(*=======================================================*)
	170:	(* WT Nummer schreiben *)
		IF	 fb_state_entry.E THEN
			(* Starte Schreib Prozess *)
			balluff_tag_reader.fb.i16_addresse := 0;
			balluff_tag_reader.fb.i16_anzahl_byte := 1;
			balluff_tag_reader.fb.s_schreib_daten[0] := gst_tag_data.WpcNumber;
			balluff_tag_reader.st_ctrl.in.b_start_schreiben := TRUE;
		END_IF

		(*-----------------------Weiterschaltbedingungen----------------------------*)
		IF 	balluff_tag_reader.st_ctrl.out.b_fertig AND NOT fb_state_entry.E THEN
			balluff_tag_reader.st_ctrl.in.b_start_schreiben := FALSE;
			fb_state_entry.i16_next_step := 180;
		END_IF

(*=======================================================*)
	180:	(* letztes benutzes Werkzeug schreiben*)
		IF 	fb_state_entry.E THEN
			(* Starte Schreib Prozess *)
			IF gst_datensatz.st_md.i16_tag_data_structur_version = 0 THEN
				balluff_tag_reader.fb.i16_addresse := 54;
				balluff_tag_reader.fb.i16_anzahl_byte := 1;
				balluff_tag_reader.fb.s_schreib_daten[0] := gst_tag_data.LastUsedTool;
				balluff_tag_reader.st_ctrl.in.b_start_schreiben := TRUE;
			ELSIF gst_datensatz.st_md.i16_tag_data_structur_version = 1 THEN
				balluff_tag_reader.fb.i16_addresse := 15;
				balluff_tag_reader.fb.i16_anzahl_byte := 1;
				balluff_tag_reader.fb.s_schreib_daten[0] := gst_tag_data.LastUsedTool;
				balluff_tag_reader.st_ctrl.in.b_start_schreiben := TRUE;
			END_IF
		END_IF

		(*-----------------------Weiterschaltbedingungen----------------------------*)
		IF 	balluff_tag_reader.st_ctrl.out.b_fertig AND NOT fb_state_entry.E THEN
			balluff_tag_reader.st_ctrl.in.b_start_schreiben := FALSE;
			IF gst_datensatz.st_md.i16_tag_data_structur_version = 0 THEN
				fb_state_entry.i16_next_step := 120;
			ELSIF gst_datensatz.st_md.i16_tag_data_structur_version = 1 THEN
				fb_state_entry.i16_next_step := 190;
			END_IF
		END_IF

(*=======================================================*)
	190:	(* Anzahl ISK auf WT *)
		IF 	fb_state_entry.E THEN
			(* Starte Schreib Prozess *)
			balluff_tag_reader.fb.i16_addresse := 10;
			balluff_tag_reader.fb.i16_anzahl_byte := 1;
			balluff_tag_reader.fb.s_schreib_daten[0] := gst_tag_data.AmountPartsOnWpc;
			balluff_tag_reader.st_ctrl.in.b_start_schreiben := TRUE;
		END_IF

		(*-----------------------Weiterschaltbedingungen----------------------------*)
		IF 	balluff_tag_reader.st_ctrl.out.b_fertig AND NOT fb_state_entry.E THEN
			balluff_tag_reader.st_ctrl.in.b_start_schreiben := FALSE;
			fb_state_entry.i16_next_step := 120;
		END_IF

(*=======================================================*)
	200:	(*WT zurücksetzen*)
		IF	 fb_state_entry.E THEN
			IF gst_datensatz.st_md.i16_tag_data_structur_version = 0 THEN
				gst_tag_data.StateParts[0] := PART_NO;
				gst_tag_data.StateParts[1] := PART_NO;

				balluff_tag_reader.st_ctrl.in.b_start_schreiben := TRUE;
				balluff_tag_reader.fb.i16_addresse := 1;
				balluff_tag_reader.fb.i16_anzahl_byte := 2;
				balluff_tag_reader.fb.s_schreib_daten[0] := DINT_TO_BYTE(gst_tag_data.StateParts[0]);
				balluff_tag_reader.fb.s_schreib_daten[1] := DINT_TO_BYTE(gst_tag_data.StateParts[1]);
			ELSIF gst_datensatz.st_md.i16_tag_data_structur_version = 1 THEN
				FOR i:= 0 TO 7 BY 1 DO
					gst_tag_data.StateParts[i] := PART_NO;
				END_FOR
	
				balluff_tag_reader.st_ctrl.in.b_start_schreiben := TRUE;
				balluff_tag_reader.fb.i16_addresse := 1;
				balluff_tag_reader.fb.i16_anzahl_byte := 8;
				FOR i:= 0 TO 7 BY 1 DO
					balluff_tag_reader.fb.s_schreib_daten[i] := DINT_TO_BYTE(gst_tag_data.StateParts[i]);
				END_FOR
			END_IF
		END_IF

		(*-----------------------Weiterschaltbedingungen----------------------------*)
		IF 	balluff_tag_reader.st_ctrl.out.b_fertig AND NOT fb_state_entry.E THEN
			(* Ok: Daten sind auf dem Tag *)
			balluff_tag_reader.st_ctrl.in.b_start_schreiben := FALSE;
			fb_state_entry.i16_next_step := 210;
		END_IF

(*=======================================================*)
	210:	(* letztes benutzes Werkzeug schreiben*)
		IF 	fb_state_entry.E THEN
			gst_tag_data.LastUsedTool := 0;
			(* Starte Schreib Prozess *)
			IF gst_datensatz.st_md.i16_tag_data_structur_version = 0 THEN
				balluff_tag_reader.fb.i16_addresse := 54;
				balluff_tag_reader.fb.i16_anzahl_byte := 1;
				balluff_tag_reader.fb.s_schreib_daten[0] := 0;
				balluff_tag_reader.st_ctrl.in.b_start_schreiben := TRUE;
			ELSIF gst_datensatz.st_md.i16_tag_data_structur_version = 1 THEN
				balluff_tag_reader.fb.i16_addresse := 15;
				balluff_tag_reader.fb.i16_anzahl_byte := 1;
				balluff_tag_reader.fb.s_schreib_daten[0] := 0;
				balluff_tag_reader.st_ctrl.in.b_start_schreiben := TRUE;
			END_IF
		END_IF

		(*-----------------------Weiterschaltbedingungen----------------------------*)
		IF 	balluff_tag_reader.st_ctrl.out.b_fertig AND NOT fb_state_entry.E THEN
			balluff_tag_reader.st_ctrl.in.b_start_schreiben := FALSE;
			fb_state_entry.i16_next_step := INIT;
		END_IF

(*=======================================================*)
	FEHLER:
		IF 	fb_state_entry.E THEN
			st_ctrl_out.b_fehler := TRUE;
			fb_ton_quitt.IN := FALSE;
		END_IF

		(*-----------------------Weiterschaltbedingungen----------------------------*)
		IF 	st_ctrl_in.b_quitt AND NOT fb_state_entry.E THEN
			st_ctrl_out.b_fehler := FALSE;
			fb_ton_quitt.IN := TRUE;
		END_IF

		IF 	fb_ton_quitt.Q THEN
			fb_ton_quitt.IN := FALSE;
			fb_state_entry.i16_next_step := INIT;
		END_IF

(*=======================================================*)
	STOP:
		IF 	fb_state_entry.E THEN
			;
		END_IF

		(*-----------------------Weiterschaltbedingungen----------------------------*)
		IF 	Balluff_Tag_Reader.fb.fb_state_entry.i16_step=BEREIT THEN
			fb_state_entry.i16_next_step := INIT;
		END_IF

END_CASE

fb_state_entry(
	i16_next_step:= ,
	i16_pos:= 2,
	s_debugtext:= ,
	E=> ,
	X=> ,
	i16_step=> ,
	i16_last_step=> );

(* Fehlermeldungen ab dem Startindex in das globale Störmeldungsarray schreiben *)
garr_stoermeldungen[st_config.i16_meld_startindex + 0] := sm_WT_Nummer_ungueltig;
garr_stoermeldungen[st_config.i16_meld_startindex + 1] := sm_wt_hat_kein_tag;
garr_stoermeldungen[st_config.i16_meld_startindex + 2] :=FALSE;
garr_stoermeldungen[st_config.i16_meld_startindex + 3] := FALSE;
garr_stoermeldungen[st_config.i16_meld_startindex + 4] := FALSE;
garr_stoermeldungen[st_config.i16_meld_startindex + 5] := FALSE;
garr_stoermeldungen[st_config.i16_meld_startindex + 6] := FALSE;
garr_stoermeldungen[st_config.i16_meld_startindex + 7] := FALSE;
garr_stoermeldungen[st_config.i16_meld_startindex + 8] := FALSE;
garr_stoermeldungen[st_config.i16_meld_startindex + 9] := FALSE;
garr_stoermeldungen[st_config.i16_meld_startindex + 10] := FALSE;
garr_stoermeldungen[st_config.i16_meld_startindex + 11] := FALSE;
garr_stoermeldungen[st_config.i16_meld_startindex + 12] := FALSE;
garr_stoermeldungen[st_config.i16_meld_startindex + 13] := FALSE;
garr_stoermeldungen[st_config.i16_meld_startindex + 14] := FALSE;
garr_stoermeldungen[st_config.i16_meld_startindex + 15] := FALSE;
garr_stoermeldungen[st_config.i16_meld_startindex + 16] := FALSE;
garr_stoermeldungen[st_config.i16_meld_startindex + 17] := FALSE;
garr_stoermeldungen[st_config.i16_meld_startindex + 18] := FALSE;
garr_stoermeldungen[st_config.i16_meld_startindex + 19] := FALSE;

garr_betriebsmeldungen[st_config.i16_meld_startindex + 0] := bm_kein_WT_im_Aktionsfeld;
garr_betriebsmeldungen[st_config.i16_meld_startindex + 1] := bm_Wert_nicht_erlaubt;
garr_betriebsmeldungen[st_config.i16_meld_startindex + 2] := FALSE;
garr_betriebsmeldungen[st_config.i16_meld_startindex + 3] := FALSE;
garr_betriebsmeldungen[st_config.i16_meld_startindex + 4] := FALSE;
garr_betriebsmeldungen[st_config.i16_meld_startindex + 5] := FALSE;
garr_betriebsmeldungen[st_config.i16_meld_startindex + 6] := FALSE;
garr_betriebsmeldungen[st_config.i16_meld_startindex + 7] := FALSE;
garr_betriebsmeldungen[st_config.i16_meld_startindex + 8] := FALSE;
garr_betriebsmeldungen[st_config.i16_meld_startindex + 9] := FALSE;
garr_betriebsmeldungen[st_config.i16_meld_startindex + 10] := FALSE;
garr_betriebsmeldungen[st_config.i16_meld_startindex + 11] := FALSE;
garr_betriebsmeldungen[st_config.i16_meld_startindex + 12] := FALSE;
garr_betriebsmeldungen[st_config.i16_meld_startindex + 13] := FALSE;
garr_betriebsmeldungen[st_config.i16_meld_startindex + 14] := FALSE;
garr_betriebsmeldungen[st_config.i16_meld_startindex + 15] := FALSE;
garr_betriebsmeldungen[st_config.i16_meld_startindex + 16] := FALSE;
garr_betriebsmeldungen[st_config.i16_meld_startindex + 17] := FALSE;
garr_betriebsmeldungen[st_config.i16_meld_startindex + 18] := FALSE;
garr_betriebsmeldungen[st_config.i16_meld_startindex + 19] := FALSE;
END_PROGRAM

(* POU Gemeinsamkeiten17xx/Bandeinzug/ST_Anwahl_Bandeinzug, ST *)
PROGRAM ST_Anwahl_Bandeinzug
VAR
	b_first_cycle 						: BOOL := TRUE;
	i16_typ_bandeinzug_visu			: enum_typ_bandeinzug_visu := KEIN_BANDEINZUG;
END_VAR
(*======================================================
   PRG: ExportResultString
 ------------------------------------------------------
   Auth: 		Werner Friedl    						 
   Date: 		07.03.2016    						     
   Rev.: 		1.0	
   Desc:		Damit bei unterschiedlichen Zellen (1700 oder 1720) nur die vorhandenen Bandwechsler in der Visu vorne angezeigt werden,
			müssen diese der Struktur "i16_typ_bandeinzug" zugewiesen werden.
   Historie:   1.0

 ========================================================*)
IF 	gi16_bbgen_auftrag = LESE_WKZ THEN
	b_first_cycle:=TRUE;
END_IF



IF	NOT b_first_cycle THEN

	CASE gst_datensatz.st_md.i16_typ_zelle OF
		KEINE_ZELLE:
			;

		BESTUECKZELLE_1700, RASTERFOLIE:
	
			CASE i16_typ_bandeinzug_visu OF

				KEIN_BANDEINZUG :
						gst_datensatz.st_wkz.i16_typ_bandeinzug:=KEIN_EINZUG;					;
				BANDEINZUG_1:
						gst_datensatz.st_wkz.i16_typ_bandeinzug:=BANDWECHSLER_V2;
				BANDEINZUG_2:
						gst_datensatz.st_wkz.i16_typ_bandeinzug:=SERVO;
				BANDEINZUG_3:
					;
			END_CASE

		BESTUECKZELLE_1720:

			CASE i16_typ_bandeinzug_visu OF
	
				KEIN_BANDEINZUG :
						gst_datensatz.st_wkz.i16_typ_bandeinzug:=KEIN_EINZUG;
				BANDEINZUG_1:
						gst_datensatz.st_wkz.i16_typ_bandeinzug:=STANDARD_2FACH_V2;
				BANDEINZUG_2:
					;
				BANDEINZUG_3:
					;
			END_CASE

	END_CASE

ELSIF	 gi16_bbgen_auftrag = KEIN_BB_AUFTRAG AND b_first_cycle THEN

	CASE gst_datensatz.st_md.i16_typ_zelle OF
		KEINE_ZELLE:
			;

		BESTUECKZELLE_1700, RASTERFOLIE:

			CASE gst_datensatz.st_wkz.i16_typ_bandeinzug OF

				KEIN_EINZUG :
					i16_typ_bandeinzug_visu:=KEIN_BANDEINZUG;
				BANDWECHSLER_V2:
					i16_typ_bandeinzug_visu:=BANDEINZUG_1;
				SERVO:
					i16_typ_bandeinzug_visu:=BANDEINZUG_2;

			END_CASE
			b_first_cycle:=FALSE;

		BESTUECKZELLE_1720:
	
			CASE gst_datensatz.st_wkz.i16_typ_bandeinzug OF

				KEIN_EINZUG :
					i16_typ_bandeinzug_visu:=KEIN_BANDEINZUG;
				STANDARD_2FACH_V2:
					i16_typ_bandeinzug_visu:=BANDEINZUG_1;

			END_CASE
			b_first_cycle:=FALSE;

	END_CASE


END_IF
END_PROGRAM

(* POU Gemeinsamkeiten17xx/Allgemeines/ST_Scope, ST *)
PROGRAM ST_Scope
VAR
	fb_ton_wz			: TON;
	fb_r_trig_bereit		: R_TRIG;
	fb_state_entry			: ST_StateEntry;

	fb_ScopeStop		: ScopeSetOffline;
	fb_ScopeOnline		: ScopeSetOnline;
	fb_ScopeExport		: ScopeViewExport;

	b_Stop				: BOOL;
	s_file_name			: STRING;
	pos					: INT;
	i					: INT;
	i32_error_id			:UDINT;
END_VAR

VAR CONSTANT
	s_path				: STRING:='C:\TwinCAT\Scope\';
END_VAR
(*===============================================================
   PRG: ST_Scope
  ---------------------------------------------------------------
   Auth: 		Werner Friedl
   Date: 		03.08.2016    						    
   Rev.: 		1.0
   Beschreibung:
	Mit diesem Programm wird das Scope automatisch gestartet und bei einem Fehler 
	ein Scopedatei mit aktueller Zeit im Verzeichnis "C:\TwinCAT\Scope\" abgespeichert. 

	-	zuerst muss ein Scope geöffnet und ein Projekt erstellt werden.
	-	Fehler für Stop eintragen	
	-	ST_ScopeStop startet das Scope bei "Anlage betriebsbereit"
	-	bei Fehler wird die Aufzeichnung nach 2sec gestoppt
	-	Auzeichnung	wird mit aktueller Zeit abgespeichert.	

hier Fehler für Stop einfügen============================================*)
(*b_Stop:=	ST_Bestueckachse.st_ctrl_out.b_fehler  OR
		axis_bestueckachse.st_ctrl.out.b_fehler ;*)

b_Stop:= (gi16_maschinenstatusinfo = STATUS_FEHLER);

(*=======================================================*)
fb_ton_wz(IN:=,PT:=T#2s);
fb_r_trig_bereit(CLK:= gi16_maschinenstatusinfo = STATUS_BETRIEBSBEREIT, Q=> );
fb_ScopeStop(bExecute:= , bBusy=> , bError=> , iErrorId=> );
fb_ScopeOnline(bExecute:= , bBusy=> , bError=> , iErrorId=> );
fb_ScopeExport(bExecute:=, sFilePath:=, tTimeout:=T#5s);

(*=======================================================*)
fb_state_entry(i16_pos:= 1, );

CASE fb_state_entry.i16_step OF
(*=======================================================*)
	INIT_OBJ:
		fb_state_entry.i16_next_step := INIT;

(*=======================================================*)
	INIT:
		IF	fb_state_entry.E THEN
			fb_ScopeOnline.bExecute:=FALSE;
			fb_ScopeStop.bExecute:=FALSE;
			fb_ScopeExport.bExecute:=FALSE;
		END_IF

		fb_state_entry.i16_next_step := BEREIT;


(*=======================================================*)
	BEREIT: (*warten auf betriebsbereit *)
		IF	fb_state_entry.E THEN
			b_Stop:=FALSE;
		END_IF

		IF	fb_r_trig_bereit.Q THEN
			fb_state_entry.i16_next_step := 110;
		END_IF


(*=======================================================*)
	110: (* Scope starten *)
		IF 	fb_state_entry.E THEN
			fb_ScopeOnline.bExecute:=TRUE;
		END_IF

		(*-----------------------Weiterschaltbedingungen----------------------------*)
		IF	fb_ScopeOnline.bBusy THEN
			fb_state_entry.i16_next_step := 120;
		END_IF

(*=======================================================*)
	120: (* Scope starten *)

		IF	NOT fb_ScopeOnline.bBusy THEN
			fb_state_entry.i16_next_step := 130;
			fb_ScopeOnline.bExecute:=FALSE;
		END_IF

		IF	fb_ScopeOnline.bError THEN
			i32_error_id:=fb_ScopeOnline.iErrorId;
			fb_state_entry.i16_next_step := FEHLER;
		END_IF

(*=======================================================*)
	130: (* warten auf Fehler *)
		IF	 fb_state_entry.E THEN
			fb_ton_wz.IN:=FALSE;
		END_IF

		fb_ton_wz.IN:=b_Stop ;
		fb_ScopeStop.bExecute:=fb_ton_wz.Q;


		IF	fb_ScopeStop.bBusy THEN
			fb_state_entry.i16_next_step := 140;
		END_IF

		IF	 fb_state_entry.X THEN
			fb_ton_wz.IN:=FALSE;
		END_IF
(*=======================================================*)
	140: (* Scope anhalten *)

		IF	NOT fb_ScopeStop.bBusy THEN
			fb_ScopeStop.bExecute:=FALSE;
			fb_state_entry.i16_next_step := 150;
		END_IF

		IF	fb_ScopeStop.bError THEN
			i32_error_id:=fb_ScopeStop.iErrorId;
			fb_state_entry.i16_next_step := FEHLER;
		END_IF

(*=======================================================*)
	150: (* Scope speichern *)
		IF 	fb_state_entry.E THEN
			s_file_name:=gstr_system_time;
			i:=0;
			FOR i := 1 TO 5  BY 1DO
				pos:=0;
				pos:=FIND(s_file_name,':');
				IF	pos > 0 THEN
					s_file_name:=REPLACE(s_file_name,'-',1,pos);
				END_IF
			END_FOR

			s_file_name:=CONCAT(s_file_name,'_Scope_View');
			s_file_name:=CONCAT(s_file_name,'.svw');

			fb_ScopeExport.sFilePath:=CONCAT(s_path,s_file_name);
			fb_ScopeExport.bExecute:=TRUE;
		END_IF

		(*-----------------------Weiterschaltbedingungen----------------------------*)
		IF	fb_ScopeExport.bBusy THEN
			fb_state_entry.i16_next_step := 160;
		END_IF


(*=======================================================*)
	160: (* Scope speichern *)

		IF	NOT fb_ScopeExport.bBusy THEN
			fb_state_entry.i16_next_step := BEREIT;
			fb_ScopeExport.bExecute:=FALSE;
		END_IF

		IF	fb_ScopeExport.bError THEN
			i32_error_id:=fb_ScopeExport.iErrorId;
			fb_state_entry.i16_next_step := FEHLER;
		END_IF

(*=======================================================*)
	FEHLER:	(*bei Fehler einfach weiter*)
		IF 	fb_state_entry.E THEN
			;
		END_IF
			fb_state_entry.i16_next_step := INIT;

END_CASE

fb_state_entry(i16_pos:= 2 );
END_PROGRAM

(* POU Maschine1720/ST_Stoerungen_Quitt_1720, ST *)
PROGRAM ST_Stoerungen_Quitt_1720
VAR_INPUT
	st_config					: struct_config;
	st_ctrl_in					: struct_ctrl_in;
END_VAR
VAR_IN_OUT
	st_visu					: struct_visu;
	st_visu_hinten				: struct_visu_hinten;
END_VAR
VAR_OUTPUT
	st_ctrl_out				: struct_ctrl_out;
	b_lampe_stoerung		: BOOL;
	b_lampe_produktion		: BOOL;
END_VAR
VAR
	fb_ton_quitt				: TON;
	fb_r_trig_quittieren			: R_TRIG;
	b_Merker_quitt			: BOOL:=FALSE;
	fb_ton_wz				: TON;

	fb_state_entry				: ST_StateEntry;

	fb_blinker				: ST_Blinker;

	bm_Maschine_in_Gst		: BOOL := FALSE;
	bm_Check		: BOOL := FALSE;
	sm_disable_auto_reset	: BOOL := FALSE;
END_VAR
(* Zeiten *)
fb_ton_quitt(IN:= , PT:= t#300ms, Q=> , ET=> );

(* Flanken *)
fb_r_trig_quittieren(CLK:= (st_visu.b_quittieren OR st_visu_hinten.out.b_quittieren) AND gi16_betriebsart <> HAND, Q=> );

(* Blinker *)
fb_blinker(
	b_start:= TRUE,
	t_taktzeit_on:=t#500ms,
	t_taktzeit_off:=t#500ms,
	b_blinker_out=> );

(* Lampen *)
b_lampe_stoerung := gi16_maschinenstatusinfo = KEIN_STATUS OR gi16_maschinenstatusinfo = STATUS_FEHLER;

b_lampe_produktion := (fb_blinker.b_blinker_out AND
					(gi16_maschinenstatusinfo = STATUS_FEHLER_QUITTIERT OR
					gi16_maschinenstatusinfo = STATUS_BETRIEBSBEREIT)) OR
					gi16_maschinenstatusinfo = STATUS_MASCHINE_ARBEITET;

bm_Check:=(
	CheckBounds_ErrCnt+
	CheckByteZeroDiv_ErrCnt+
	CheckDWordZeroDiv_ErrCnt+
	CheckRealZeroDiv_ErrCnt+
	CheckWordZeroDiv_ErrCnt+
	CheckRangeSigned_ErrCnt+
	CheckRangeUnsigned_ErrCnt) > 0 ;

(* Toplevel *)
(* Hier nur Abschaltungen welche zu sofortigem Stop führen müssen *)
IF fb_state_entry.i16_step < FEHLER AND
	(axis_virt_master.st_ctrl.out.b_fehler OR
	axis_bestueckachse.st_ctrl.out.b_fehler OR
	axis_z_achse.st_ctrl.out.b_fehler OR
	bandeinzug_kontroller.st_ctrl.out.b_fehler OR
	bandspruehoeler.st_ctrl.out.b_fehler OR
	wkz_absicherung.st_ctrl.out.b_fehler OR
	wt_transport_kontroller.st_ctrl.out.b_fehler OR
(*	hublift_links.st_ctrl.out.b_fehler OR
	hublift_rechts.st_ctrl.out.b_fehler OR*)
	balluff_tag_reader.st_ctrl.out.b_fehler OR
	haspel_kontroller.st_ctrl.out.b_fehler OR
	bbgen.st_ctrl.out.b_fehler OR
	wartung.st_ctrl.out.b_fehler OR
	betriebsfreigaben.st_ctrl.out.b_fehler OR
	safety.st_ctrl.out.b_fehler OR
	edit_mfps.st_ctrl.out.b_fehler OR
	Lesen_Schreiben_Tag.st_ctrl.out.b_fehler OR
	Service.st_ctrl.out.b_fehler)
	THEN
		fb_state_entry.i16_next_step := FEHLER;
END_IF

(* Prüfe ob BA = Hand -> Stoppe Abläufe *)
IF  fb_state_entry.i16_step > INIT  AND fb_state_entry.i16_step < FEHLER  AND gi16_betriebsart = HAND THEN
	fb_state_entry.i16_next_step := FEHLER;
END_IF

(* ======================================Schrittkette======================================== *)
fb_state_entry(
	i16_next_step:= ,
	i16_pos:= 1,
	s_debugtext:= ,
	E=> ,
	X=> ,
	i16_step=> ,
	i16_last_step=> );

CASE fb_state_entry.i16_step OF
(*=======================================================*)
	INIT_OBJ:
		IF st_config.b_config_fertig THEN
			fb_state_entry.i16_next_step := FEHLER;
		END_IF

(*=======================================================*)
	INIT:
		IF fb_state_entry.E THEN
			gi16_maschinenstatusinfo := STATUS_FEHLER_QUITTIERT;

			fb_ton_quitt.IN := FALSE;
			UPS.st_ctrl.in.b_quitt := FALSE;
			betriebsfreigaben.st_ctrl.in.b_quitt := FALSE;
			bandeinzug_kontroller.st_ctrl.in.b_quitt := FALSE;
			axis_virt_master.st_ctrl.in.b_quitt := FALSE;
			axis_bestueckachse.st_ctrl.in.b_quitt := FALSE;
			axis_z_achse.st_ctrl.in.b_quitt := FALSE;
			bandspruehoeler.st_ctrl.in.b_quitt := FALSE;
			haspel_kontroller.st_ctrl.in.b_quitt := FALSE;
			hublift_links.st_ctrl.in.b_quitt := FALSE;
			hublift_rechts.st_ctrl.in.b_quitt := FALSE;
			wt_transport_kontroller.st_ctrl.in.b_quitt := FALSE;
			wkz_absicherung.st_ctrl.in.b_quitt := FALSE;
			stueckzahlen.st_ctrl.in.b_quitt := FALSE;
			balluff_tag_reader.st_ctrl.in.b_quitt := FALSE;
			bbgen.st_ctrl.in.b_quitt := FALSE;
			wartung.st_ctrl.in.b_quitt := FALSE;
			safety.st_ctrl.in.b_quitt := FALSE;
			edit_mfps.st_ctrl.in.b_quitt := FALSE;
			routing_backpanel.st_ctrl.in.b_quitt := FALSE;
			routing_nachbarpc.st_ctrl.in.b_quitt := FALSE;
			bm_Maschine_in_Gst := FALSE;
			Lesen_Schreiben_Tag.st_ctrl.in.b_quitt :=FALSE;
			Service.st_ctrl.in.b_quitt :=FALSE;
			ST_TippTasten.b_initialisierungsphase := TRUE;
			sm_disable_auto_reset := FALSE;
		END_IF

		(*-----------------------Weiterschaltbedingungen----------------------------*)
		IF safety.st_ctrl.out.b_bereit THEN
			fb_state_entry.i16_next_step := 11;
		END_IF

(*=======================================================*)
	11:
		IF fb_state_entry.E THEN
			axis_virt_master.st_ctrl.in.b_preinit := TRUE;
		END_IF

		(*-----------------------Weiterschaltbedingungen----------------------------*)
		IF axis_virt_master.st_ctrl.out.b_prebereit  THEN
			axis_virt_master.st_ctrl.in.b_preinit := FALSE;
			fb_state_entry.i16_next_step := 12;
		END_IF

(*=======================================================*)
	12:
		IF fb_state_entry.E THEN
			axis_z_achse.st_ctrl.in.b_preinit := TRUE;
		END_IF

		(*-----------------------Weiterschaltbedingungen----------------------------*)
		IF axis_z_achse.st_ctrl.out.b_prebereit  THEN
			axis_z_achse.st_ctrl.in.b_preinit := FALSE;
			fb_state_entry.i16_next_step := 14;
		END_IF

(*=======================================================*)
	14:
		IF fb_state_entry.E THEN
			axis_bestueckachse.st_ctrl.in.b_preinit := TRUE;
		END_IF

		(*-----------------------Weiterschaltbedingungen----------------------------*)
		IF axis_bestueckachse.st_ctrl.out.b_prebereit THEN
			axis_bestueckachse.st_ctrl.in.b_preinit := FALSE;
			fb_state_entry.i16_next_step := 16;
		END_IF

(*=======================================================*)
	16:
		(*Wenn die Bestückachse nicht in einem bestimmten Bereich steht, dann muss sie von Hand
		    freigefahren werden. Außer es ist die Nocke auf 0,0 gestellt*)
		IF	gst_datensatz.st_wkz.nockenschaltwerk_bestueckachse.arr_nocken[SP_DISABLE_AUTO_RESET].r_cam_begin = 0 AND
			gst_datensatz.st_wkz.nockenschaltwerk_bestueckachse.arr_nocken[SP_DISABLE_AUTO_RESET].r_cam_end = 0 THEN
				fb_state_entry.i16_next_step := 20;
		ELSE
			IF gst_datensatz.st_wkz.nockenschaltwerk_bestueckachse.arr_nocken[SP_DISABLE_AUTO_RESET].r_cam_begin > gst_datensatz.st_wkz.nockenschaltwerk_bestueckachse.arr_nocken[SP_DISABLE_AUTO_RESET].r_cam_end THEN
				IF bestueckachse.NcToPlc.ModuloActPos > gst_datensatz.st_wkz.nockenschaltwerk_bestueckachse.arr_nocken[SP_DISABLE_AUTO_RESET].r_cam_begin OR
					bestueckachse.NcToPlc.ModuloActPos < gst_datensatz.st_wkz.nockenschaltwerk_bestueckachse.arr_nocken[SP_DISABLE_AUTO_RESET].r_cam_end THEN
					sm_disable_auto_reset := TRUE;
					fb_state_entry.i16_next_step := FEHLER;
				ELSE
					fb_state_entry.i16_next_step := 20;
				END_IF
			ELSE
				IF bestueckachse.NcToPlc.ModuloActPos > gst_datensatz.st_wkz.nockenschaltwerk_bestueckachse.arr_nocken[SP_DISABLE_AUTO_RESET].r_cam_begin AND
					bestueckachse.NcToPlc.ModuloActPos < gst_datensatz.st_wkz.nockenschaltwerk_bestueckachse.arr_nocken[SP_DISABLE_AUTO_RESET].r_cam_end THEN
					sm_disable_auto_reset := TRUE;
					fb_state_entry.i16_next_step := FEHLER;
				ELSE
					fb_state_entry.i16_next_step := 20;
				END_IF
			END_IF
		END_IF

(*=======================================================*)
	20:
		IF fb_state_entry.E THEN
			haspel_kontroller.st_ctrl.in.b_init := TRUE;
			bandspruehoeler.st_ctrl.in.b_init := TRUE;
			wkz_absicherung.st_ctrl.in.b_init := TRUE;
			stueckzahlen.st_ctrl.in.b_init := TRUE;
			(*balluff_tag_reader.st_ctrl.in.b_init := TRUE;*)
			edit_mfps.st_ctrl.in.b_init := TRUE;
		END_IF

		(*-----------------------Weiterschaltbedingungen----------------------------*)
		IF 	haspel_kontroller.st_ctrl.out.b_bereit  AND
			bandspruehoeler.st_ctrl.out.b_bereit  AND
			wkz_absicherung.st_ctrl.out.b_bereit AND
			balluff_tag_reader.st_ctrl.out.b_bereit AND
			edit_mfps.st_ctrl.out.b_bereit
			THEN
				haspel_kontroller.st_ctrl.in.b_init := FALSE;
				bandspruehoeler.st_ctrl.in.b_init := FALSE;
				wkz_absicherung.st_ctrl.in.b_init := FALSE;
				stueckzahlen.st_ctrl.in.b_init := FALSE;
				(*balluff_tag_reader.st_ctrl.in.b_init := FALSE;*)
				edit_mfps.st_ctrl.in.b_init := FALSE;
				fb_state_entry.i16_next_step := 30;
		END_IF

(*=======================================================*)
	30:
		IF fb_state_entry.E THEN
			bandeinzug_kontroller.st_ctrl.in.b_init := TRUE;
		END_IF

		(*-----------------------Weiterschaltbedingungen----------------------------*)
		IF bandeinzug_kontroller.st_ctrl.out.b_bereit THEN
			bandeinzug_kontroller.st_ctrl.in.b_init := FALSE;
			fb_state_entry.i16_next_step := 40;
		END_IF

(*=======================================================*)
	40:
		IF fb_state_entry.E THEN
			axis_bestueckachse.st_ctrl.in.b_init := TRUE;
		END_IF

		(*-----------------------Weiterschaltbedingungen----------------------------*)
		IF axis_bestueckachse.st_ctrl.out.b_bereit  THEN
			axis_bestueckachse.st_ctrl.in.b_init := FALSE;
			fb_state_entry.i16_next_step := 50;
		END_IF

(*=======================================================*)
	50:
		IF fb_state_entry.E THEN
			axis_z_achse.st_ctrl.in.b_init := TRUE;
		END_IF

		(*-----------------------Weiterschaltbedingungen----------------------------*)
		IF axis_z_achse.st_ctrl.out.b_bereit THEN
			axis_z_achse.st_ctrl.in.b_init := FALSE;
			fb_state_entry.i16_next_step := 60;
		END_IF

(*=======================================================*)
	60:
		IF fb_state_entry.E THEN
			axis_virt_master.st_ctrl.in.b_init := TRUE;
		END_IF

		(*-----------------------Weiterschaltbedingungen----------------------------*)
		IF axis_virt_master.st_ctrl.out.b_bereit  THEN
			axis_virt_master.st_ctrl.in.b_init := FALSE;
			fb_state_entry.i16_next_step := 70;
		END_IF

(*=======================================================*)
	70:
		IF fb_state_entry.E THEN
			hublift_links.st_ctrl.in.b_init := TRUE;
			hublift_rechts.st_ctrl.in.b_init := TRUE;
			wt_transport_kontroller.st_ctrl.in.b_init := TRUE;
		END_IF

		(*-----------------------Weiterschaltbedingungen----------------------------*)
		IF hublift_links.st_ctrl.out.b_bereit AND hublift_rechts.st_ctrl.out.b_bereit AND wt_transport_kontroller.st_ctrl.out.b_bereit THEN
			hublift_links.st_ctrl.in.b_init := FALSE;
			hublift_rechts.st_ctrl.in.b_init := FALSE;
			wt_transport_kontroller.st_ctrl.in.b_init := FALSE;
			fb_state_entry.i16_next_step := BEREIT;
		END_IF

(*=======================================================*)
	BEREIT:
		IF fb_state_entry.E THEN
			ST_TippTasten.b_initialisierungsphase  := FALSE;

			(* Setze Maschinenstatus *)
			bm_Maschine_in_Gst := TRUE;
		END_IF

		(*Beim Einfädeln muss der Status geändert werden, damit nicht
		ständig neue Maschinendaten erzeugt werden*)
		IF ST_TippTasten.b_einfaedeln_aktiv THEN
			gi16_maschinenstatusinfo := STATUS_MASCHINE_ARBEITET;
		ELSE
			gi16_maschinenstatusinfo := STATUS_BETRIEBSBEREIT;
		END_IF

		(*-----------------------Weiterschaltbedingungen----------------------------*)
		IF NOT wt_transport_kontroller.st_ctrl.out.b_fertig THEN
			bm_Maschine_in_Gst := FALSE;
			fb_state_entry.i16_next_step := 110;
		END_IF

(*=======================================================*)
	110: (* Produktion *)
		IF fb_state_entry.E THEN
			gi16_maschinenstatusinfo := STATUS_MASCHINE_ARBEITET;
		END_IF

		(*-----------------------Weiterschaltbedingungen----------------------------*)
		IF wt_transport_kontroller.st_ctrl.out.b_fertig THEN
			fb_state_entry.i16_next_step := BEREIT;
		END_IF

(*=======================================================*)
	FEHLER:
		IF fb_state_entry.E THEN
			gi16_maschinenstatusinfo := STATUS_FEHLER;
			bm_Maschine_in_Gst := FALSE;
			ST_TippTasten.b_initialisierungsphase  := FALSE;
			fb_ton_quitt.IN := FALSE;
			fb_ton_wz.IN:=FALSE;
			s_alte_artikelnummer := '';

			(* Schlecht Stueckzahl erhöhen *)
			IF fb_state_entry.i16_last_step = 110 THEN
				stueckzahlen.st_ctrl.in.b_schlechtteil_produziert := TRUE;
			END_IF

			UPS.st_ctrl.in.b_quitt := FALSE;
			betriebsfreigaben.st_ctrl.in.b_quitt := FALSE;
			bandeinzug_kontroller.st_ctrl.in.b_quitt := FALSE;
			axis_virt_master.st_ctrl.in.b_quitt := FALSE;
			axis_bestueckachse.st_ctrl.in.b_quitt := FALSE;
			axis_z_achse.st_ctrl.in.b_quitt := FALSE;
			bandspruehoeler.st_ctrl.in.b_quitt := FALSE;
			haspel_kontroller.st_ctrl.in.b_quitt := FALSE;
			hublift_links.st_ctrl.in.b_quitt := FALSE;
			hublift_rechts.st_ctrl.in.b_quitt := FALSE;
			wt_transport_kontroller.st_ctrl.in.b_quitt := FALSE;
			wkz_absicherung.st_ctrl.in.b_quitt := FALSE;
			stueckzahlen.st_ctrl.in.b_quitt := FALSE;
			balluff_tag_reader.st_ctrl.in.b_quitt := FALSE;
			bbgen.st_ctrl.in.b_quitt := FALSE;
			wartung.st_ctrl.in.b_quitt := FALSE;
			safety.st_ctrl.in.b_quitt := FALSE;
			edit_mfps.st_ctrl.in.b_quitt := FALSE;
			routing_backpanel.st_ctrl.in.b_quitt := FALSE;
			routing_nachbarpc.st_ctrl.in.b_quitt := FALSE;
			Lesen_Schreiben_Tag.st_ctrl.in.b_quitt := FALSE;
			Service.st_ctrl.in.b_quitt := FALSE;

			axis_virt_master.st_ctrl.in.b_preinit := FALSE;
			axis_bestueckachse.st_ctrl.in.b_preinit := FALSE;
			axis_z_achse.st_ctrl.in.b_preinit := FALSE;

			bandeinzug_kontroller.st_ctrl.in.b_init := FALSE;
			axis_virt_master.st_ctrl.in.b_init := FALSE;
			axis_bestueckachse.st_ctrl.in.b_init := FALSE;
			axis_z_achse.st_ctrl.in.b_init := FALSE;
			bandspruehoeler.st_ctrl.in.b_init := FALSE;
			haspel_kontroller.st_ctrl.in.b_init := FALSE;
			hublift_links.st_ctrl.in.b_init := FALSE;
			hublift_rechts.st_ctrl.in.b_init := FALSE;
			wt_transport_kontroller.st_ctrl.in.b_init := FALSE;
			wkz_absicherung.st_ctrl.in.b_init := FALSE;
			stueckzahlen.st_ctrl.in.b_init := FALSE;
			balluff_tag_reader.st_ctrl.in.b_init := FALSE;
			edit_mfps.st_ctrl.in.b_init := FALSE;
		END_IF

		(* Fehlerhandling: was soll bei welchem Fehler passieren? *)
		IF 	NOT fb_ton_quitt.IN THEN
			(* Stoppe/Halte Komponenten an *)
			bandeinzug_kontroller.st_ctrl.in.b_stop := TRUE;
			bandspruehoeler.st_ctrl.in.b_stop := TRUE;
			(*haspel_kontroller.st_ctrl.in.b_stop := TRUE;*)
			hublift_links.st_ctrl.in.b_stop := TRUE;
			hublift_rechts.st_ctrl.in.b_stop := TRUE;
			wt_transport_kontroller.st_ctrl.in.b_stop := TRUE;
			stueckzahlen.st_ctrl.in.b_stop := TRUE;
			balluff_tag_reader.st_ctrl.in.b_stop := TRUE;
			edit_mfps.st_ctrl.in.b_stop := TRUE;

			(* Diese Fehler führt zum "Stop" in der Maschine *)
			IF safety.st_ctrl.out.b_fehler THEN
				axis_virt_master.st_ctrl.in.b_stop := TRUE;
				axis_bestueckachse.st_ctrl.in.b_stop := TRUE;
				axis_z_achse.st_ctrl.in.b_stop := TRUE;
				axis_virt_master.st_ctrl.in.b_halt := FALSE;
				axis_bestueckachse.st_ctrl.in.b_halt := FALSE;
				axis_z_achse.st_ctrl.in.b_halt := FALSE;
			ELSE
				axis_virt_master.st_ctrl.in.b_halt := TRUE;
				axis_bestueckachse.st_ctrl.in.b_halt := TRUE;
				axis_z_achse.st_ctrl.in.b_halt := TRUE;
				axis_virt_master.st_ctrl.in.b_stop := FALSE;
				axis_bestueckachse.st_ctrl.in.b_stop := FALSE;
				axis_z_achse.st_ctrl.in.b_stop := FALSE;
			END_IF
		END_IF

		(*-----------------------Weiterschaltbedingungen----------------------------*)
		IF 	fb_r_trig_quittieren.Q THEN
			fb_ton_wz.IN:=TRUE;
			b_Merker_quitt:=TRUE;
		END_IF
		IF 	(b_Merker_quitt AND ST_Betriebsfreigaben.e_druckwaechter) OR
			fb_ton_wz.Q THEN
			fb_ton_wz.IN:=FALSE;
			b_Merker_quitt:=FALSE;
			fb_ton_quitt.IN := TRUE;
			(* QUITT *)
			UPS.st_ctrl.in.b_quitt := TRUE;
			betriebsfreigaben.st_ctrl.in.b_quitt := TRUE;
			bandeinzug_kontroller.st_ctrl.in.b_quitt := TRUE;
			axis_virt_master.st_ctrl.in.b_quitt := TRUE;
			axis_bestueckachse.st_ctrl.in.b_quitt := TRUE;
			axis_z_achse.st_ctrl.in.b_quitt := TRUE;
			bandspruehoeler.st_ctrl.in.b_quitt := TRUE;
			haspel_kontroller.st_ctrl.in.b_quitt := TRUE;
			hublift_links.st_ctrl.in.b_quitt := TRUE;
			hublift_rechts.st_ctrl.in.b_quitt := TRUE;
			wt_transport_kontroller.st_ctrl.in.b_quitt := TRUE;
			wkz_absicherung.st_ctrl.in.b_quitt := TRUE;
			stueckzahlen.st_ctrl.in.b_quitt := TRUE;
			balluff_tag_reader.st_ctrl.in.b_quitt := TRUE;
			bbgen.st_ctrl.in.b_quitt := TRUE;
			wartung.st_ctrl.in.b_quitt := TRUE;
			safety.st_ctrl.in.b_quitt := TRUE;
			edit_mfps.st_ctrl.in.b_quitt := TRUE;
			routing_backpanel.st_ctrl.in.b_quitt := TRUE;
			routing_nachbarpc.st_ctrl.in.b_quitt := TRUE;
			Lesen_Schreiben_Tag.st_ctrl.in.b_quitt := TRUE;
			Service.st_ctrl.in.b_quitt := TRUE;
			(* STOP *)
			bandeinzug_kontroller.st_ctrl.in.b_stop := FALSE;
			axis_virt_master.st_ctrl.in.b_stop := FALSE;
			axis_bestueckachse.st_ctrl.in.b_stop := FALSE;
			axis_z_achse.st_ctrl.in.b_stop := FALSE;
			bandspruehoeler.st_ctrl.in.b_stop := FALSE;
			haspel_kontroller.st_ctrl.in.b_stop := FALSE;
			hublift_links.st_ctrl.in.b_stop := FALSE;
			hublift_rechts.st_ctrl.in.b_stop := FALSE;
			wt_transport_kontroller.st_ctrl.in.b_stop := FALSE;
			wkz_absicherung.st_ctrl.in.b_stop := FALSE;
			stueckzahlen.st_ctrl.in.b_stop := FALSE;
			balluff_tag_reader.st_ctrl.in.b_stop := FALSE;
			edit_mfps.st_ctrl.in.b_stop := FALSE;
			(* HALT - nur Achsen *)
			axis_virt_master.st_ctrl.in.b_halt := FALSE;
			axis_bestueckachse.st_ctrl.in.b_halt := FALSE;
			axis_z_achse.st_ctrl.in.b_halt := FALSE;
		END_IF

		IF fb_ton_quitt.Q THEN
			IF (gi16_betriebsart = AUTO OR gi16_betriebsart = TIPPEN) THEN
				fb_state_entry.i16_next_step := INIT;
			END_IF
		END_IF
END_CASE

fb_state_entry(
	i16_next_step:= ,
	i16_pos:= 2,
	s_debugtext:= ,
	E=> ,
	X=> , 
	i16_step=> ,
	i16_last_step=> );

IF st_config.b_config_fertig THEN
	(* Fehlermeldungen und Betriebsmeldungen ab dem Startindex in die globalen Meldungsarrays schreiben *)
	garr_stoermeldungen[st_config.i16_meld_startindex + 0] := sm_disable_auto_reset;
	garr_stoermeldungen[st_config.i16_meld_startindex + 1] := FALSE;
	garr_stoermeldungen[st_config.i16_meld_startindex + 2] := FALSE;
	garr_stoermeldungen[st_config.i16_meld_startindex + 3] := FALSE;
	garr_stoermeldungen[st_config.i16_meld_startindex + 4] := FALSE;
	garr_stoermeldungen[st_config.i16_meld_startindex + 5] := FALSE;
	garr_stoermeldungen[st_config.i16_meld_startindex + 6] := FALSE;
	garr_stoermeldungen[st_config.i16_meld_startindex + 7] := FALSE;
	garr_stoermeldungen[st_config.i16_meld_startindex + 8] := FALSE;
	garr_stoermeldungen[st_config.i16_meld_startindex + 9] := FALSE;
	garr_stoermeldungen[st_config.i16_meld_startindex + 10] := FALSE;
	garr_stoermeldungen[st_config.i16_meld_startindex + 11] := FALSE;
	garr_stoermeldungen[st_config.i16_meld_startindex + 12] := FALSE;
	garr_stoermeldungen[st_config.i16_meld_startindex + 13] := FALSE;
	garr_stoermeldungen[st_config.i16_meld_startindex + 14] := FALSE;
	garr_stoermeldungen[st_config.i16_meld_startindex + 15] := FALSE;
	garr_stoermeldungen[st_config.i16_meld_startindex + 16] := FALSE;
	garr_stoermeldungen[st_config.i16_meld_startindex + 17] := FALSE;
	garr_stoermeldungen[st_config.i16_meld_startindex + 18] := FALSE;
	garr_stoermeldungen[st_config.i16_meld_startindex + 19] := FALSE;
	
	garr_betriebsmeldungen[st_config.i16_meld_startindex + 0] := bm_Maschine_in_Gst;
	garr_betriebsmeldungen[st_config.i16_meld_startindex + 1] := bm_Check;
	garr_betriebsmeldungen[st_config.i16_meld_startindex + 2] := FALSE;
	garr_betriebsmeldungen[st_config.i16_meld_startindex + 3] := FALSE;
	garr_betriebsmeldungen[st_config.i16_meld_startindex + 4] := FALSE;
	garr_betriebsmeldungen[st_config.i16_meld_startindex + 5] := FALSE;
	garr_betriebsmeldungen[st_config.i16_meld_startindex + 6] := FALSE;
	garr_betriebsmeldungen[st_config.i16_meld_startindex + 7] := FALSE;
	garr_betriebsmeldungen[st_config.i16_meld_startindex + 8] := FALSE;
	garr_betriebsmeldungen[st_config.i16_meld_startindex + 9] := FALSE;
	garr_betriebsmeldungen[st_config.i16_meld_startindex + 10] := FALSE;
	garr_betriebsmeldungen[st_config.i16_meld_startindex + 11] := FALSE;
	garr_betriebsmeldungen[st_config.i16_meld_startindex + 12] := FALSE;
	garr_betriebsmeldungen[st_config.i16_meld_startindex + 13] := FALSE;
	garr_betriebsmeldungen[st_config.i16_meld_startindex + 14] := FALSE;
	garr_betriebsmeldungen[st_config.i16_meld_startindex + 15] := FALSE;
	garr_betriebsmeldungen[st_config.i16_meld_startindex + 16] := FALSE;
	garr_betriebsmeldungen[st_config.i16_meld_startindex + 17] := FALSE;
	garr_betriebsmeldungen[st_config.i16_meld_startindex + 18] := FALSE;
	garr_betriebsmeldungen[st_config.i16_meld_startindex + 19] := FALSE;
END_IF
END_PROGRAM

(* POU Maschine1720/ST_AbfallBlasluft, ST *)
PROGRAM ST_AbfallBlasluft
VAR_INPUT
	b_wkz_blasluft_aktiv	: BOOL;
END_VAR
VAR
	a_AbfallBlasluft		AT %Q* : BOOL;
	fb_rtrig_nocke		: R_TRIG;
	fb_tof_blaszeit		: TOF;
	b_blasluft_aktiv		: BOOL := FALSE;
END_VAR
fb_rtrig_nocke (CLK:= (bestueckachse.NcToPlc.ModuloActPos > 170 AND bestueckachse.NcToPlc.ModuloActPos < 190), Q=> );

IF b_wkz_blasluft_aktiv THEN
	fb_tof_blaszeit (IN:=fb_rtrig_nocke.Q , PT:= t#200ms, Q=> a_AbfallBlasluft, ET=> );
END_IF
END_PROGRAM

(* POU Rasterfolie/ST_Rafl_Stoerungen_Quitt, ST *)
PROGRAM ST_Rafl_Stoerungen_Quitt
VAR_INPUT
	st_config						: struct_config;
	st_ctrl_in						: struct_ctrl_in;
END_VAR
VAR_IN_OUT
	st_visu						: struct_visu;
	st_visu_hinten					: struct_visu_hinten;
END_VAR
VAR_OUTPUT
	st_ctrl_out					: struct_ctrl_out;
	b_lampe_stoerung			: BOOL;
	b_lampe_produktion			: BOOL;
END_VAR
VAR
	fb_ton_quitt					: TON;
	fb_ton_wz				: TON;
	fb_r_trig_quittieren				: R_TRIG;
	fb_state_entry					: ST_StateEntry;

	fb_blinker					: ST_Blinker;
	b_Merker_quitt			: BOOL:=FALSE;
	bm_Maschine_in_Gst			: BOOL := FALSE;
END_VAR
(* Zeiten *)
fb_ton_quitt(IN:= , PT:= t#150ms, Q=> , ET=> );
fb_ton_wz(IN:= , PT:= t#3000ms, Q=> , ET=> );

(* Flanken *)
fb_r_trig_quittieren(CLK:= (st_visu.b_quittieren OR st_visu_hinten.out.b_quittieren) AND gi16_betriebsart <> HAND, Q=> );

(* Blinker *)
fb_blinker(
	b_start:= TRUE,
	t_taktzeit_on:=t#500ms,
	t_taktzeit_off:=t#500ms,
	b_blinker_out=> );

(* Lampen *)
b_lampe_stoerung := gi16_maschinenstatusinfo = KEIN_STATUS OR gi16_maschinenstatusinfo = STATUS_FEHLER;

b_lampe_produktion := (fb_blinker.b_blinker_out AND
					(gi16_maschinenstatusinfo = STATUS_FEHLER_QUITTIERT OR
					gi16_maschinenstatusinfo = STATUS_BETRIEBSBEREIT)) OR
					gi16_maschinenstatusinfo = STATUS_MASCHINE_ARBEITET;

(* Toplevel *)
(* Hier nur Abschaltungen welche zu sofortigem Stop führen müssen *)
IF fb_state_entry.i16_step < FEHLER AND
	(axis_virt_master.st_ctrl.out.b_fehler OR
	axis_bestueckachse.st_ctrl.out.b_fehler OR
	axis_z_achse.st_ctrl.out.b_fehler OR
	axis_y_achse.st_ctrl.out.b_fehler OR
	ST_TouchProbe.st_ctrl_out.b_fehler OR
	haspel_kontroller.st_ctrl.out.b_fehler OR
	rasterfolieneinzug.st_ctrl.out.b_fehler OR
	rasterfolienmontage.st_ctrl.out.b_fehler OR
	wt_transport_kontroller.st_ctrl.out.b_fehler OR
	balluff_tag_reader.st_ctrl.out.b_fehler OR
	bbgen.st_ctrl.out.b_fehler OR
	betriebsfreigaben.st_ctrl.out.b_fehler OR
	safety.st_ctrl.out.b_fehler OR
	edit_mfps.st_ctrl.out.b_fehler OR
	Lesen_Schreiben_Tag.st_ctrl.out.b_fehler OR
	Service.st_ctrl.out.b_fehler)
	THEN
		fb_state_entry.i16_next_step := FEHLER;
END_IF

(* Prüfe ob BA = Hand -> Stoppe Abläufe *)
IF  fb_state_entry.i16_step > INIT  AND fb_state_entry.i16_step < FEHLER  AND gi16_betriebsart = HAND THEN
	fb_state_entry.i16_next_step := FEHLER;
END_IF

(* ======================================Schrittkette======================================== *)
fb_state_entry(
	i16_next_step:= ,
	i16_pos:= 1,
	s_debugtext:= ,
	E=> ,
	X=> ,
	i16_step=> ,
	i16_last_step=> );

CASE fb_state_entry.i16_step OF
(*=======================================================*)
	INIT_OBJ:
		IF st_config.b_config_fertig THEN
			fb_state_entry.i16_next_step := FEHLER;
		END_IF

(*=======================================================*)
	INIT:
		IF fb_state_entry.E THEN
			gi16_maschinenstatusinfo := STATUS_FEHLER_QUITTIERT;
			fb_ton_quitt.IN := FALSE;
			betriebsfreigaben.st_ctrl.in.b_quitt := FALSE;
			safety.st_ctrl.in.b_quitt := FALSE;
			rasterfolienmontage.st_ctrl.in.b_quitt := FALSE;
			rasterfolieneinzug.st_ctrl.in.b_quitt := FALSE;
			axis_virt_master.st_ctrl.in.b_quitt := FALSE;
			axis_bestueckachse.st_ctrl.in.b_quitt := FALSE;
			axis_y_achse.st_ctrl.in.b_quitt := FALSE;
			axis_z_achse.st_ctrl.in.b_quitt := FALSE;
			ST_TouchProbe.st_ctrl_in.b_quitt := FALSE;
			hublift_links.st_ctrl.in.b_quitt := FALSE;
			hublift_rechts.st_ctrl.in.b_quitt := FALSE;
			stueckzahlen.st_ctrl.in.b_quitt := FALSE;
			wt_transport_kontroller.st_ctrl.in.b_quitt := FALSE;
			balluff_tag_reader.st_ctrl.in.b_quitt := FALSE;
			bbgen.st_ctrl.in.b_quitt := FALSE;
			edit_mfps.st_ctrl.in.b_quitt := FALSE;
			routing_backpanel.st_ctrl.in.b_quitt := FALSE;
			routing_nachbarpc.st_ctrl.in.b_quitt := FALSE;
			bm_Maschine_in_Gst := FALSE;
			Lesen_Schreiben_Tag.st_ctrl.in.b_quitt := FALSE;
			Service.st_ctrl.in.b_quitt := FALSE;
			ST_TippTasten.b_initialisierungsphase  := TRUE;
			haspel_kontroller.st_ctrl.in.b_quitt := FALSE;
		END_IF

		(*-----------------------Weiterschaltbedingungen----------------------------*)
		IF safety.st_ctrl.out.b_bereit THEN
			fb_state_entry.i16_next_step := 11;
		END_IF

(*=======================================================*)
	11:
		IF fb_state_entry.E THEN
			axis_virt_master.st_ctrl.in.b_preinit := TRUE;
		END_IF

		(*-----------------------Weiterschaltbedingungen----------------------------*)
		IF axis_virt_master.st_ctrl.out.b_prebereit  THEN
			axis_virt_master.st_ctrl.in.b_preinit := FALSE;
			fb_state_entry.i16_next_step := 12;
		END_IF

(*=======================================================*)
	12:
		IF fb_state_entry.E THEN
			axis_z_achse.st_ctrl.in.b_preinit := TRUE;
		END_IF

		(*-----------------------Weiterschaltbedingungen----------------------------*)
		IF axis_z_achse.st_ctrl.out.b_prebereit  THEN
			axis_z_achse.st_ctrl.in.b_preinit := FALSE;
			fb_state_entry.i16_next_step := 14;
		END_IF

(*=======================================================*)
	14:
		IF fb_state_entry.E THEN
			axis_y_achse.st_ctrl.in.b_preinit := TRUE;
		END_IF

		(*-----------------------Weiterschaltbedingungen----------------------------*)
		IF axis_y_achse.st_ctrl.out.b_prebereit  THEN
			axis_y_achse.st_ctrl.in.b_preinit := FALSE;
			fb_state_entry.i16_next_step := 16;
		END_IF

(*=======================================================*)
	16:
		IF fb_state_entry.E THEN
			axis_bestueckachse.st_ctrl.in.b_preinit := TRUE;
		END_IF

		(*-----------------------Weiterschaltbedingungen----------------------------*)
		IF axis_bestueckachse.st_ctrl.out.b_prebereit THEN
			axis_bestueckachse.st_ctrl.in.b_preinit := FALSE;
			fb_state_entry.i16_next_step := 20;
		END_IF

(*=======================================================*)
	20:
		IF fb_state_entry.E THEN
			haspel_kontroller.st_ctrl.in.b_init := TRUE;
			stueckzahlen.st_ctrl.in.b_init := TRUE;
			balluff_tag_reader.st_ctrl.in.b_init := TRUE;
			rasterfolienmontage.st_ctrl.in.b_init := TRUE;
			edit_mfps.st_ctrl.in.b_init := TRUE;
		END_IF

		(*-----------------------Weiterschaltbedingungen----------------------------*)
		IF	haspel_kontroller.st_ctrl.out.b_bereit AND
			rasterfolienmontage.st_ctrl.out.b_bereit AND
			balluff_tag_reader.st_ctrl.out.b_bereit AND
			edit_mfps.st_ctrl.out.b_bereit
			THEN
				haspel_kontroller.st_ctrl.in.b_init := FALSE;
				stueckzahlen.st_ctrl.in.b_init := FALSE;
				balluff_tag_reader.st_ctrl.in.b_init := FALSE;
				rasterfolienmontage.st_ctrl.in.b_init := FALSE;
				edit_mfps.st_ctrl.in.b_init := FALSE;
				fb_state_entry.i16_next_step := 30;
		END_IF

(*=======================================================*)
	30:
		IF fb_state_entry.E THEN
			rasterfolieneinzug.st_ctrl.in.b_init := TRUE;
		END_IF

		(*-----------------------Weiterschaltbedingungen----------------------------*)
		IF rasterfolieneinzug.st_ctrl.out.b_bereit THEN
			rasterfolieneinzug.st_ctrl.in.b_init := FALSE;
			fb_state_entry.i16_next_step := 40;
		END_IF

(*=======================================================*)
	40:
		IF fb_state_entry.E THEN
			axis_bestueckachse.st_ctrl.in.b_init := TRUE;
		END_IF

		(*-----------------------Weiterschaltbedingungen----------------------------*)
		IF axis_bestueckachse.st_ctrl.out.b_bereit  THEN
			axis_bestueckachse.st_ctrl.in.b_init := FALSE;
			fb_state_entry.i16_next_step := 50;
		END_IF

(*=======================================================*)
	50:
		IF fb_state_entry.E THEN
			axis_z_achse.st_ctrl.in.b_init := TRUE;
			axis_y_achse.st_ctrl.in.b_init := TRUE;
		END_IF

		(*-----------------------Weiterschaltbedingungen----------------------------*)
		IF axis_z_achse.st_ctrl.out.b_bereit AND axis_y_achse.st_ctrl.out.b_bereit THEN
			axis_z_achse.st_ctrl.in.b_init := FALSE;
			axis_y_achse.st_ctrl.in.b_init := FALSE;
			fb_state_entry.i16_next_step := 60;
		END_IF

(*=======================================================*)
	60:
		IF fb_state_entry.E THEN
			axis_virt_master.st_ctrl.in.b_init := TRUE;
		END_IF

		(*-----------------------Weiterschaltbedingungen----------------------------*)
		IF axis_virt_master.st_ctrl.out.b_bereit  THEN
			axis_virt_master.st_ctrl.in.b_init := FALSE;
			fb_state_entry.i16_next_step := 70;
		END_IF

(*=======================================================*)
	70:
		IF fb_state_entry.E THEN
			hublift_links.st_ctrl.in.b_init := TRUE;
			hublift_rechts.st_ctrl.in.b_init := TRUE;
			wt_transport_kontroller.st_ctrl.in.b_init := TRUE;
			ST_TouchProbe.st_ctrl_in.b_init := TRUE;
		END_IF

		(*-----------------------Weiterschaltbedingungen----------------------------*)
		IF 	hublift_links.st_ctrl.out.b_bereit AND
			hublift_rechts.st_ctrl.out.b_bereit AND
			wt_transport_kontroller.st_ctrl.out.b_bereit AND
			ST_TouchProbe.st_ctrl_out.b_bereit
			THEN
				hublift_links.st_ctrl.in.b_init := FALSE;
				hublift_rechts.st_ctrl.in.b_init := FALSE;
				wt_transport_kontroller.st_ctrl.in.b_init := FALSE;
				ST_TouchProbe.st_ctrl_in.b_init := FALSE;
				fb_state_entry.i16_next_step := BEREIT;
		END_IF

(*=======================================================*)
	BEREIT:
		IF fb_state_entry.E THEN
			ST_TippTasten.b_initialisierungsphase  := FALSE;

			(* Setze Maschinenstatus *)
			bm_Maschine_in_Gst := TRUE;
		END_IF

		(*Beim Einfädeln muss der Status geändert werden, damit nicht
		ständig neue Maschinendaten erzeugt werden*)
		IF ST_TippTasten.b_einfaedeln_aktiv THEN
			gi16_maschinenstatusinfo := STATUS_MASCHINE_ARBEITET;
		ELSE
			gi16_maschinenstatusinfo := STATUS_BETRIEBSBEREIT;
		END_IF

		(*-----------------------Weiterschaltbedingungen----------------------------*)
		IF NOT wt_transport_kontroller.st_ctrl.out.b_fertig THEN
			bm_Maschine_in_Gst := FALSE;
			fb_state_entry.i16_next_step := 110;
		END_IF

(*=======================================================*)
	110: (* Produktion *)
		IF fb_state_entry.E THEN
			gi16_maschinenstatusinfo := STATUS_MASCHINE_ARBEITET;
		END_IF

		(*-----------------------Weiterschaltbedingungen----------------------------*)
		IF wt_transport_kontroller.st_ctrl.out.b_fertig THEN
			fb_state_entry.i16_next_step := BEREIT;
		END_IF

(*=======================================================*)
	FEHLER:
		IF fb_state_entry.E THEN
			gi16_maschinenstatusinfo := STATUS_FEHLER;
			bm_Maschine_in_Gst := FALSE;
			ST_TippTasten.b_initialisierungsphase  := FALSE;
			fb_ton_quitt.IN := FALSE;
			s_alte_artikelnummer := '';

			(* Schlecht Stueckzahl erhöhen *)
			IF fb_state_entry.i16_last_step = 110 THEN
				stueckzahlen.st_ctrl.in.b_schlechtteil_produziert := TRUE;
			END_IF

			betriebsfreigaben.st_ctrl.in.b_quitt := FALSE;
			safety.st_ctrl.in.b_quitt := FALSE;
			rasterfolienmontage.st_ctrl.in.b_quitt := FALSE;
			rasterfolieneinzug.st_ctrl.in.b_quitt := FALSE;
			axis_virt_master.st_ctrl.in.b_quitt := FALSE;
			axis_bestueckachse.st_ctrl.in.b_quitt := FALSE;
			axis_y_achse.st_ctrl.in.b_quitt := FALSE;
			axis_z_achse.st_ctrl.in.b_quitt := FALSE;
			ST_TouchProbe.st_ctrl_in.b_quitt := FALSE;
			haspel_kontroller.st_ctrl.in.b_quitt := FALSE;
			hublift_links.st_ctrl.in.b_quitt := FALSE;
			hublift_rechts.st_ctrl.in.b_quitt := FALSE;
			wt_transport_kontroller.st_ctrl.in.b_quitt := FALSE;
			stueckzahlen.st_ctrl.in.b_quitt := FALSE;
			balluff_tag_reader.st_ctrl.in.b_quitt := FALSE;
			bbgen.st_ctrl.in.b_quitt := FALSE;
			edit_mfps.st_ctrl.in.b_quitt := FALSE;
			routing_backpanel.st_ctrl.in.b_quitt := FALSE;
			routing_nachbarpc.st_ctrl.in.b_quitt := FALSE;
			Lesen_Schreiben_Tag.st_ctrl.in.b_quitt := FALSE;
			Service.st_ctrl.in.b_quitt := FALSE;

			axis_virt_master.st_ctrl.in.b_preinit := FALSE;
			axis_bestueckachse.st_ctrl.in.b_preinit := FALSE;
			axis_y_achse.st_ctrl.in.b_preinit := FALSE;
			axis_z_achse.st_ctrl.in.b_preinit := FALSE;

			rasterfolienmontage.st_ctrl.in.b_init := FALSE;
			rasterfolieneinzug.st_ctrl.in.b_init := FALSE;
			axis_virt_master.st_ctrl.in.b_init := FALSE;
			axis_bestueckachse.st_ctrl.in.b_init := FALSE;
			axis_y_achse.st_ctrl.in.b_init := FALSE;
			axis_z_achse.st_ctrl.in.b_init := FALSE;
			ST_TouchProbe.st_ctrl_in.b_init := FALSE;
			haspel_kontroller.st_ctrl.in.b_init := FALSE;
			hublift_links.st_ctrl.in.b_init := FALSE;
			hublift_rechts.st_ctrl.in.b_init := FALSE;
			wt_transport_kontroller.st_ctrl.in.b_init := FALSE;
			stueckzahlen.st_ctrl.in.b_init := FALSE;
			balluff_tag_reader.st_ctrl.in.b_init := FALSE;
			edit_mfps.st_ctrl.in.b_init := FALSE;
		END_IF

		(* Fehlerhandling: was soll bei welchem Fehler passieren? *)
		IF 	NOT fb_ton_quitt.IN THEN
			(* Stoppe/Halte Komponenten an *)
			rasterfolienmontage.st_ctrl.in.b_stop := TRUE;
			rasterfolieneinzug.st_ctrl.in.b_stop := TRUE;
			hublift_links.st_ctrl.in.b_stop := TRUE;
			hublift_rechts.st_ctrl.in.b_stop := TRUE;
			wt_transport_kontroller.st_ctrl.in.b_stop := TRUE;
			stueckzahlen.st_ctrl.in.b_stop := TRUE;
			balluff_tag_reader.st_ctrl.in.b_stop := TRUE;
			edit_mfps.st_ctrl.in.b_stop := TRUE;

			(* Diese Fehler führt zum "Stop" in der Maschine *)
			IF safety.st_ctrl.out.b_fehler THEN
				axis_virt_master.st_ctrl.in.b_stop := TRUE;
				axis_bestueckachse.st_ctrl.in.b_stop := TRUE;
				axis_z_achse.st_ctrl.in.b_stop := TRUE;
				axis_y_achse.st_ctrl.in.b_stop := TRUE;
				axis_virt_master.st_ctrl.in.b_halt := FALSE;
				axis_bestueckachse.st_ctrl.in.b_halt := FALSE;
				axis_z_achse.st_ctrl.in.b_halt := FALSE;
				axis_y_achse.st_ctrl.in.b_halt := FALSE;
			ELSE
				axis_virt_master.st_ctrl.in.b_halt := TRUE;
				axis_bestueckachse.st_ctrl.in.b_halt := TRUE;
				axis_z_achse.st_ctrl.in.b_halt := TRUE;
				axis_y_achse.st_ctrl.in.b_halt := TRUE;
				axis_virt_master.st_ctrl.in.b_stop := FALSE;
				axis_bestueckachse.st_ctrl.in.b_stop := FALSE;
				axis_z_achse.st_ctrl.in.b_stop := FALSE;
				axis_y_achse.st_ctrl.in.b_stop := FALSE;
			END_IF
		END_IF


		(*-----------------------Weiterschaltbedingungen----------------------------*)
		IF fb_r_trig_quittieren.Q THEN
			fb_ton_wz.IN:=TRUE;
			b_Merker_quitt:=TRUE;
		END_IF
		IF 	(b_Merker_quitt AND ST_Betriebsfreigaben.e_druckwaechter) OR
			fb_ton_wz.Q THEN
			fb_ton_wz.IN:=FALSE;
			b_Merker_quitt:=FALSE;
			fb_ton_quitt.IN := TRUE;
			(* QUITT *)
			betriebsfreigaben.st_ctrl.in.b_quitt := TRUE;
			safety.st_ctrl.in.b_quitt := TRUE;
			rasterfolienmontage.st_ctrl.in.b_quitt := TRUE;
			rasterfolieneinzug.st_ctrl.in.b_quitt := TRUE;
			axis_virt_master.st_ctrl.in.b_quitt := TRUE;
			axis_bestueckachse.st_ctrl.in.b_quitt := TRUE;
			axis_y_achse.st_ctrl.in.b_quitt := TRUE;
			axis_z_achse.st_ctrl.in.b_quitt := TRUE;
			ST_TouchProbe.st_ctrl_in.b_quitt := TRUE;
			haspel_kontroller.st_ctrl.in.b_quitt := TRUE;
			hublift_links.st_ctrl.in.b_quitt := TRUE;
			hublift_rechts.st_ctrl.in.b_quitt := TRUE;
			wt_transport_kontroller.st_ctrl.in.b_quitt := TRUE;
			stueckzahlen.st_ctrl.in.b_quitt := TRUE;
			balluff_tag_reader.st_ctrl.in.b_quitt := TRUE;
			bbgen.st_ctrl.in.b_quitt := TRUE;
			edit_mfps.st_ctrl.in.b_quitt := TRUE;
			routing_backpanel.st_ctrl.in.b_quitt := TRUE;
			routing_nachbarpc.st_ctrl.in.b_quitt := TRUE;
			Lesen_Schreiben_Tag.st_ctrl.in.b_quitt := TRUE;
			Service.st_ctrl.in.b_quitt := TRUE;
			(* STOP *)
			rasterfolienmontage.st_ctrl.in.b_stop := FALSE;
			rasterfolieneinzug.st_ctrl.in.b_stop := FALSE;
			axis_virt_master.st_ctrl.in.b_stop := FALSE;
			axis_bestueckachse.st_ctrl.in.b_stop := FALSE;
			axis_y_achse.st_ctrl.in.b_stop := FALSE;
			axis_z_achse.st_ctrl.in.b_stop := FALSE;
			haspel_kontroller.st_ctrl.in.b_stop := FALSE;
			hublift_links.st_ctrl.in.b_stop := FALSE;
			hublift_rechts.st_ctrl.in.b_stop := FALSE;
			wt_transport_kontroller.st_ctrl.in.b_stop := FALSE;
			stueckzahlen.st_ctrl.in.b_stop := FALSE;
			balluff_tag_reader.st_ctrl.in.b_stop := FALSE;
			edit_mfps.st_ctrl.in.b_stop := FALSE;
			(* HALT - nur Achsen *)
			axis_virt_master.st_ctrl.in.b_halt := FALSE;
			axis_bestueckachse.st_ctrl.in.b_halt := FALSE;
			axis_y_achse.st_ctrl.in.b_halt := FALSE;
			axis_z_achse.st_ctrl.in.b_halt := FALSE;
		END_IF

		IF fb_ton_quitt.Q THEN
			IF (gi16_betriebsart = AUTO OR gi16_betriebsart = TIPPEN) THEN
				fb_state_entry.i16_next_step := INIT;
			END_IF
		END_IF
END_CASE

fb_state_entry(
	i16_next_step:= ,
	i16_pos:= 2,
	s_debugtext:= ,
	E=> ,
	X=> , 
	i16_step=> ,
	i16_last_step=> );

IF st_config.b_config_fertig THEN
	(* Fehlermeldungen und Betriebsmeldungen ab dem Startindex in die globalen Meldungsarrays schreiben *)
	garr_stoermeldungen[st_config.i16_meld_startindex + 0] := FALSE;
	garr_stoermeldungen[st_config.i16_meld_startindex + 1] := FALSE;
	garr_stoermeldungen[st_config.i16_meld_startindex + 2] := FALSE;
	garr_stoermeldungen[st_config.i16_meld_startindex + 3] := FALSE;
	garr_stoermeldungen[st_config.i16_meld_startindex + 4] := FALSE;
	garr_stoermeldungen[st_config.i16_meld_startindex + 5] := FALSE;
	garr_stoermeldungen[st_config.i16_meld_startindex + 6] := FALSE;
	garr_stoermeldungen[st_config.i16_meld_startindex + 7] := FALSE;
	garr_stoermeldungen[st_config.i16_meld_startindex + 8] := FALSE;
	garr_stoermeldungen[st_config.i16_meld_startindex + 9] := FALSE;
	garr_stoermeldungen[st_config.i16_meld_startindex + 10] := FALSE;
	garr_stoermeldungen[st_config.i16_meld_startindex + 11] := FALSE;
	garr_stoermeldungen[st_config.i16_meld_startindex + 12] := FALSE;
	garr_stoermeldungen[st_config.i16_meld_startindex + 13] := FALSE;
	garr_stoermeldungen[st_config.i16_meld_startindex + 14] := FALSE;
	garr_stoermeldungen[st_config.i16_meld_startindex + 15] := FALSE;
	garr_stoermeldungen[st_config.i16_meld_startindex + 16] := FALSE;
	garr_stoermeldungen[st_config.i16_meld_startindex + 17] := FALSE;
	garr_stoermeldungen[st_config.i16_meld_startindex + 18] := FALSE;
	garr_stoermeldungen[st_config.i16_meld_startindex + 19] := FALSE;
	
	garr_betriebsmeldungen[st_config.i16_meld_startindex + 0] := bm_Maschine_in_Gst;
	garr_betriebsmeldungen[st_config.i16_meld_startindex + 1] := FALSE;
	garr_betriebsmeldungen[st_config.i16_meld_startindex + 2] := FALSE;
	garr_betriebsmeldungen[st_config.i16_meld_startindex + 3] := FALSE;
	garr_betriebsmeldungen[st_config.i16_meld_startindex + 4] := FALSE;
	garr_betriebsmeldungen[st_config.i16_meld_startindex + 5] := FALSE;
	garr_betriebsmeldungen[st_config.i16_meld_startindex + 6] := FALSE;
	garr_betriebsmeldungen[st_config.i16_meld_startindex + 7] := FALSE;
	garr_betriebsmeldungen[st_config.i16_meld_startindex + 8] := FALSE;
	garr_betriebsmeldungen[st_config.i16_meld_startindex + 9] := FALSE;
	garr_betriebsmeldungen[st_config.i16_meld_startindex + 10] := FALSE;
	garr_betriebsmeldungen[st_config.i16_meld_startindex + 11] := FALSE;
	garr_betriebsmeldungen[st_config.i16_meld_startindex + 12] := FALSE;
	garr_betriebsmeldungen[st_config.i16_meld_startindex + 13] := FALSE;
	garr_betriebsmeldungen[st_config.i16_meld_startindex + 14] := FALSE;
	garr_betriebsmeldungen[st_config.i16_meld_startindex + 15] := FALSE;
	garr_betriebsmeldungen[st_config.i16_meld_startindex + 16] := FALSE;
	garr_betriebsmeldungen[st_config.i16_meld_startindex + 17] := FALSE;
	garr_betriebsmeldungen[st_config.i16_meld_startindex + 18] := FALSE;
	garr_betriebsmeldungen[st_config.i16_meld_startindex + 19] := FALSE;
END_IF
END_PROGRAM

(* POU Gemeinsamkeiten17xx/Oeler/ST_DoppelRollenbandoeler, ST *)
PROGRAM ST_Doppelrollenbandoeler
VAR_INPUT
	st_config						: struct_config;
	st_ctrl_in						: struct_ctrl_in;
	b_ot_spur					: BOOL;
END_VAR
VAR_IN_OUT
	st_visu						: struct_oeler_visu;
	st_oelerdaten					: struct_oeler_daten;
END_VAR
VAR_OUTPUT
	st_ctrl_out					: struct_ctrl_out;
	b_oelmangel					: BOOL;
END_VAR
VAR
	fb_ton_quitt					: TON;
	dt_datum_uhrzeit_letzte_oelung	: DT;
	fb_state_entry					: ST_StateEntry;
	t_delta_zeitraum				: TIME := t#5h;
	sm_fuellstand_oeler			: BOOL := FALSE;
	fb_ton_oelzeit					: TON;
	fb_r_trig_start_oelen			: R_TRIG;
	fb_r_trig_hubimpuls			: R_TRIG;
	b_ibn_handoelen				: BOOL := FALSE;
	bm_fuellstand_oeler			: BOOL := FALSE;
	a_ventil_rolle_li	 			AT %Q* : BOOL;
	a_ventil_rolle_re	 			AT %Q* : BOOL;
	e_fuellstand					AT %I* : BOOL;
END_VAR
(* Bandöler mit Füllstandsabfrage und Zwangs- und Stillstandsölung *)
(* Oeler Impuls generieren *)
fb_ton_oelzeit(IN:= , PT:= , Q=> , ET=> );
fb_ton_quitt(IN:= , PT:= t#100ms, Q=> , ET=> );

(* Hubimpuls *)
fb_r_trig_hubimpuls(CLK:= b_ot_spur, Q=> );

(* =======================================Toplevel========================================== *)
IF fb_state_entry.i16_next_step > INIT AND fb_state_entry.i16_next_step < FEHLER THEN
	IF fb_state_entry.i16_next_step < STOP THEN
		IF st_ctrl_in.b_stop THEN
			fb_state_entry.i16_next_step := STOP;
		END_IF
	END_IF
END_IF

(* Orangene Lampe an Ampel leuchtet bei Ölbehälter leer *)
b_oelmangel := bm_fuellstand_oeler;

(* =======================================Toplevel========================================== *)
IF fb_state_entry.i16_next_step > INIT AND fb_state_entry.i16_next_step < FEHLER THEN
	IF fb_state_entry.i16_next_step < STOP THEN
		IF st_ctrl_in.b_stop THEN
			fb_state_entry.i16_next_step := STOP;
		END_IF
	END_IF
END_IF

(* Prüfe auf neue Intervalvorgabe *)
IF st_config.b_station_aktiv AND st_oelerdaten.i32_neue_intervallvorgabe <> st_oelerdaten.i32_alte_intervallvorgabe THEN
	st_oelerdaten.i32_alte_intervallvorgabe := st_oelerdaten.i32_neue_intervallvorgabe;
	st_oelerdaten.i32_aktueller_stand := st_oelerdaten.i32_neue_intervallvorgabe;
END_IF

(* ==================================Schrittkette================================ *)
fb_state_entry(
	i16_next_step:= , 
	i16_pos:= 1,
	s_debugtext:= ,
	E=> ,
	X=> , 
	i16_step=> ,
	i16_last_step=> );

CASE fb_state_entry.i16_step OF
(*=======================================================*)
	INIT_OBJ:
		IF st_config.b_config_fertig THEN
			fb_state_entry.i16_next_step := INIT;
		END_IF
		
(*=======================================================*)
	INIT:
		IF fb_state_entry.E THEN
			st_ctrl_out.b_fehler := FALSE;
			st_ctrl_out.b_bereit := FALSE;
			st_ctrl_out.b_fertig := FALSE;
			fb_ton_oelzeit.IN := FALSE;
			fb_ton_quitt.IN := FALSE;
			a_ventil_rolle_li := FALSE;
			a_ventil_rolle_re := FALSE;
			sm_fuellstand_oeler := FALSE;
			bm_fuellstand_oeler := FALSE;
		END_IF

		(*-----------------------Weiterschaltbedingungen----------------------------*)
		IF st_ctrl_in.b_init THEN
			IF st_config.b_station_aktiv THEN
				fb_state_entry.i16_next_step := 20;
			ELSE
				fb_state_entry.i16_next_step := BEREIT;
			END_IF
		END_IF

(*=======================================================*)
	20: (* Abfrage Datum / Uhrzeit wegen Ölen nach Stillstand*)

		(*-----------------------Weiterschaltbedingungen----------------------------*)
		IF (gdt_system_time - dt_datum_uhrzeit_letzte_oelung) > t_delta_zeitraum THEN
			fb_ton_oelzeit.PT := st_oelerdaten.t_oelzeit_nach_stillstand;
			fb_state_entry.i16_next_step := 30;
		ELSE
			fb_state_entry.i16_next_step := BEREIT;
		END_IF

(*=======================================================*)
	30: (* Ölen nach Stillstand *)
		IF fb_state_entry.E THEN
			dt_datum_uhrzeit_letzte_oelung := gdt_system_time;	(* Merken, dass geölt wurde *)
			fb_ton_oelzeit.IN := TRUE;
			a_ventil_rolle_li := TRUE;
			a_ventil_rolle_re := TRUE;
		END_IF

		(*-----------------------Weiterschaltbedingungen----------------------------*)
		IF  fb_ton_oelzeit.Q THEN
			fb_ton_oelzeit.IN := FALSE;
			a_ventil_rolle_li := FALSE;
			a_ventil_rolle_re := FALSE;
			fb_state_entry.i16_next_step := BEREIT;
		END_IF

(*=======================================================*)
	BEREIT:
		IF fb_state_entry.E THEN
			st_ctrl_out.b_bereit := TRUE;
		END_IF

		IF st_config.b_station_aktiv THEN
			(* Zähle Hübe *)
			IF fb_r_trig_hubimpuls.Q THEN
				(* Von der Intervallvorgabe wird runter gezählt bis Null. Dann kommt der Ölimpuls *)
				st_oelerdaten.i32_aktueller_stand := st_oelerdaten.i32_aktueller_stand - 1;
			END_IF
			(* Überwachung Füllstand *)
			IF NOT e_fuellstand THEN
				sm_fuellstand_oeler := TRUE;
				fb_state_entry.i16_next_step := FEHLER;
			END_IF

			(*-----------------------Weiterschaltbedingungen----------------------------*)
			IF  st_oelerdaten.i32_aktueller_stand <= 0 OR st_visu.b_handoelen OR b_ibn_handoelen THEN
				st_visu.b_handoelen := FALSE;
				fb_ton_oelzeit.PT := st_oelerdaten.t_ventiloeffnungszeit;
				fb_state_entry.i16_next_step := 110;
			END_IF
		END_IF

(*=======================================================*)
	110: (* Ölen *)
		IF fb_state_entry.E THEN
			dt_datum_uhrzeit_letzte_oelung := gdt_system_time;	(* Merken wann das letze mal geölt wurde *)
			IF st_oelerdaten.i32_neue_intervallvorgabe <= 0 THEN
				 st_oelerdaten.i32_neue_intervallvorgabe := 100;	(* Verhindere Dauerölung, wenn in den WKZ-Ölerdaten noch 0 drin steht *)
			END_IF
			st_oelerdaten.i32_aktueller_stand := st_oelerdaten.i32_neue_intervallvorgabe;
			fb_ton_oelzeit.IN := TRUE;
			a_ventil_rolle_li := TRUE;
			a_ventil_rolle_re := TRUE;
		END_IF

		(* Zähle Hübe *)
		IF fb_r_trig_hubimpuls.Q THEN
			(* Von der Intervallvorgabe wird runter gezählt bis Null. Dann kommt der Ölimpuls *)
			st_oelerdaten.i32_aktueller_stand := st_oelerdaten.i32_aktueller_stand - 1;
		END_IF

		(*-----------------------Weiterschaltbedingungen----------------------------*)
		IF  fb_ton_oelzeit.Q THEN
			fb_ton_oelzeit.IN := FALSE;
			a_ventil_rolle_li := FALSE;
			a_ventil_rolle_re := FALSE;
			fb_state_entry.i16_next_step := BEREIT;
		END_IF

(*=======================================================*)
	FEHLER:
		IF fb_state_entry.E THEN
			st_ctrl_out.b_fehler := TRUE;
			a_ventil_rolle_li := FALSE;
			a_ventil_rolle_re := FALSE;
			fb_ton_quitt.IN := FALSE;
		END_IF

		(*-----------------------Weiterschaltbedingungen----------------------------*)
		IF st_ctrl_in.b_quitt AND NOT fb_state_entry.E THEN
			st_ctrl_out.b_fehler := FALSE;
			fb_ton_quitt.IN := TRUE;
		END_IF

		IF fb_ton_quitt.Q THEN
			fb_ton_quitt.IN := FALSE;
			fb_state_entry.i16_next_step := INIT;
		END_IF

(*=======================================================*)
	STOP:
		IF fb_state_entry.E THEN
			a_ventil_rolle_li := FALSE;
			a_ventil_rolle_re := FALSE;
			fb_ton_quitt.IN := FALSE;
		END_IF

		(*-----------------------Weiterschaltbedingungen----------------------------*)
		IF st_ctrl_in.b_quitt AND NOT fb_state_entry.E THEN
			fb_ton_quitt.IN := TRUE;
		END_IF

		IF fb_ton_quitt.Q THEN
			fb_ton_quitt.IN := FALSE;
			fb_state_entry.i16_next_step := INIT;
		END_IF
END_CASE

fb_state_entry(
	i16_next_step:= , 
	i16_pos:= 2,
	s_debugtext:= ,
	E=> ,
	X=> , 
	i16_step=> ,
	i16_last_step=> );

IF st_config.b_config_fertig THEN
	(* Fehlermeldungen und Betriebsmeldungen ab dem Startindex in die globalen Meldungsarrays schreiben *)
	garr_stoermeldungen[st_config.i16_meld_startindex + 0] := sm_fuellstand_oeler;
	garr_stoermeldungen[st_config.i16_meld_startindex + 1] := FALSE;
	garr_stoermeldungen[st_config.i16_meld_startindex + 2] := FALSE;
	garr_stoermeldungen[st_config.i16_meld_startindex + 3] := FALSE;
	garr_stoermeldungen[st_config.i16_meld_startindex + 4] := FALSE;
	garr_stoermeldungen[st_config.i16_meld_startindex + 5] := FALSE;
	garr_stoermeldungen[st_config.i16_meld_startindex + 6] := FALSE;
	garr_stoermeldungen[st_config.i16_meld_startindex + 7] := FALSE;
	garr_stoermeldungen[st_config.i16_meld_startindex + 8] := FALSE;
	garr_stoermeldungen[st_config.i16_meld_startindex + 9] := FALSE;
	garr_stoermeldungen[st_config.i16_meld_startindex + 10] := FALSE;
	garr_stoermeldungen[st_config.i16_meld_startindex + 11] := FALSE;
	garr_stoermeldungen[st_config.i16_meld_startindex + 12] := FALSE;
	garr_stoermeldungen[st_config.i16_meld_startindex + 13] := FALSE;
	garr_stoermeldungen[st_config.i16_meld_startindex + 14] := FALSE;
	garr_stoermeldungen[st_config.i16_meld_startindex + 15] := FALSE;
	garr_stoermeldungen[st_config.i16_meld_startindex + 16] := FALSE;
	garr_stoermeldungen[st_config.i16_meld_startindex + 17] := FALSE;
	garr_stoermeldungen[st_config.i16_meld_startindex + 18] := FALSE;
	garr_stoermeldungen[st_config.i16_meld_startindex + 19] := FALSE;
	
	garr_betriebsmeldungen[st_config.i16_meld_startindex + 0] := bm_fuellstand_oeler;
	garr_betriebsmeldungen[st_config.i16_meld_startindex + 1] := FALSE;
	garr_betriebsmeldungen[st_config.i16_meld_startindex + 2] := FALSE;
	garr_betriebsmeldungen[st_config.i16_meld_startindex + 3] := FALSE;
	garr_betriebsmeldungen[st_config.i16_meld_startindex + 4] := FALSE;
	garr_betriebsmeldungen[st_config.i16_meld_startindex + 5] := FALSE;
	garr_betriebsmeldungen[st_config.i16_meld_startindex + 6] := FALSE;
	garr_betriebsmeldungen[st_config.i16_meld_startindex + 7] := FALSE;
	garr_betriebsmeldungen[st_config.i16_meld_startindex + 8] := FALSE;
	garr_betriebsmeldungen[st_config.i16_meld_startindex + 9] := FALSE;
	garr_betriebsmeldungen[st_config.i16_meld_startindex + 10] := FALSE;
	garr_betriebsmeldungen[st_config.i16_meld_startindex + 11] := FALSE;
	garr_betriebsmeldungen[st_config.i16_meld_startindex + 12] := FALSE;
	garr_betriebsmeldungen[st_config.i16_meld_startindex + 13] := FALSE;
	garr_betriebsmeldungen[st_config.i16_meld_startindex + 14] := FALSE;
	garr_betriebsmeldungen[st_config.i16_meld_startindex + 15] := FALSE;
	garr_betriebsmeldungen[st_config.i16_meld_startindex + 16] := FALSE;
	garr_betriebsmeldungen[st_config.i16_meld_startindex + 17] := FALSE;
	garr_betriebsmeldungen[st_config.i16_meld_startindex + 18] := FALSE;
	garr_betriebsmeldungen[st_config.i16_meld_startindex + 19] := FALSE;
END_IF
END_PROGRAM

(* POU Maschine1700/Einpresskraftueberwachung/ST_Einpress_Kontroller_alt, ST *)
PROGRAM ST_Einpress_Kontroller_alt
VAR_INPUT
	st_config									: struct_config;
	st_ctrl_in									: struct_ctrl_in;
	lr_achsposition							: LREAL;
END_VAR
VAR_IN_OUT
	st_visu									: struct_visu;
	st_einpressen							: struct_einpresskraftueberwachung;
END_VAR
VAR_OUTPUT
	st_ctrl_out								: struct_ctrl_out;
END_VAR
VAR
	fb_ton_wz								: TON;
	fb_ton_uez								: TON;
	fb_ton_quitt								: TON;
	fb_r_trig_start								: R_TRIG;
	fb_state_entry								: ST_StateEntry;
	lr_kraft_n									: LREAL := 0.0;
	lr_weg_grad								: LREAL := 0.0;
	i16_pin_nr								: INT := 0;
	i16_kraftfaktor								: INT := 0;
	ui_akt_pos_bestueckachse					: UINT := 0;
	i16_ku_nr								: INT := 0;
	i16_mp_nr								: INT := 0;
	b_kraft_weg_in_mp_ok						: BOOL := FALSE;
	sm_fehler_einpressmodus					: BOOL := FALSE;
	sm_aktkraft_groesser_maxkraft_aufnahme	: BOOL := FALSE;
	sm_aktkraft_groesser_maxkraft_einpressen	: BOOL := FALSE;
	sm_aktkraft_kleiner_minkraft_einpressen		: BOOL := FALSE;
	sm_kraft_weg_ausserhalb_huellkurve		: BOOL := FALSE;
	sm_fehler_analogwert_kraftmessdose		: BOOL := FALSE;
	sm_max_mb_ueberschritten					: BOOL := FALSE;
	sm_max_einstell_mb_ueberschritten			: BOOL := FALSE;

	a_start_messung							AT %Q* : BOOL := FALSE;
	a_messbereich_1_oder_2					AT %Q* : BOOL := FALSE;	(* MB1 = low, MB2 = high *)

	st_ausgabe								: struct_einpressausgabe;
	i16_merker								: INT := 0;
	lr_help_maxkraft_einpressen				:LREAL;
END_VAR
VAR CONSTANT
	i_KRAFTFAKTOR_MB1		: INT := 200;	(* Der Kraftfaktor richtet sich nach der Messbereichskalibrierung in der Zusatzsoftware (ICAM) für den Ladungsverstärker *)
	i_KRAFTFAKTOR_MB2		: INT := 2000;
	i_MAX_MESSPUNKTE			: INT := 360;
	i_MAX_KURVEN				: INT := 99;
END_VAR
(* Zeiten *)
fb_ton_wz(IN:= , PT:= , Q=>  , ET=> );
fb_ton_uez(IN:= , PT:= , Q=>  , ET=> );

fb_ton_quitt(IN:= , PT:= t#100ms, Q=> , ET=> );

(* Flanken *)
fb_r_trig_start(CLK:= st_ctrl_in.b_start, Q=> );

(* Analogwert Kraftmessdose *)
kraftmessdose.fb(
	t_verzoegerung:= t#500ms,
	st_config:= kraftmessdose.fb.st_config);

(* Berechnung der aktuellen Kraft in Newton aus dem Analogwert in  Volt. *)
(* Die Normierung der Analogspannung als Kraft erfolgt mit dem Kalibrierschein der Kraftmessdose und der Software "ICAM5073" *)
(* Eingestellter Messbereich1: 0 - 200N, Messbereich2: 0 - 2000N *)
IF a_messbereich_1_oder_2 THEN
	i16_kraftfaktor := i_KRAFTFAKTOR_MB2;
ELSE
	i16_kraftfaktor := i_KRAFTFAKTOR_MB1;
END_IF

(* nur bei voller Drehzahl mit eingestellter Kraft prüfen*)
IF	ST_TippTasten.i16_akt_stufe = 9 THEN
	lr_help_maxkraft_einpressen:=st_einpressen.st_einstellungen.lr_maxkraft_einpressen;
ELSE
	lr_help_maxkraft_einpressen:=800;
END_IF

(* Behandlung Ausnahmefall Division durch 0  *)
IF kraftmessdose.fb.i16_anzeigewert_max <> 0 THEN
	lr_kraft_n := i16_kraftfaktor * kraftmessdose.fb.st_sensor.e_i16_value / kraftmessdose.fb.i16_anzeigewert_max;
END_IF

lr_weg_grad := lr_achsposition;
ui_akt_pos_bestueckachse := LREAL_TO_UINT(lr_achsposition);

(* ===============Toplevel================ *)
IF fb_state_entry.i16_next_step > INIT AND fb_state_entry.i16_next_step < FEHLER THEN
	IF fb_state_entry.i16_next_step < STOP THEN
		IF st_ctrl_in.b_stop THEN
			fb_state_entry.i16_next_step := STOP;
		END_IF
	END_IF

	(* Fehlersignal der Kraftmessdose *)
	IF st_config.b_station_aktiv THEN
		IF kraftmessdose.fb.b_error THEN
			sm_fehler_analogwert_kraftmessdose := TRUE;
			fb_state_entry.i16_next_step := FEHLER;
		END_IF
		IF 	(NOT a_messbereich_1_oder_2 AND lr_kraft_n > i_KRAFTFAKTOR_MB1) OR
			(a_messbereich_1_oder_2 AND lr_kraft_n > i_KRAFTFAKTOR_MB2) OR
			(gst_datensatz.st_band.st_einpressen.st_einstellungen.lr_maxkraft_einpressen > i_KRAFTFAKTOR_MB2)
			THEN
				sm_max_mb_ueberschritten := TRUE;
				fb_state_entry.i16_next_step := FEHLER;
		END_IF
		IF gst_datensatz.st_band.st_einpressen.st_einstellungen.lr_maxkraft_einpressen > i_KRAFTFAKTOR_MB2 THEN
			sm_max_einstell_mb_ueberschritten := TRUE;
			fb_state_entry.i16_next_step := FEHLER;
		END_IF
	END_IF
END_IF

(* ======================================Schrittkette======================================== *)
fb_state_entry(
	i16_next_step:= ,
	i16_pos:= 1,
	s_debugtext:= ,
	E=> ,
	X=> ,
	i16_step=> ,
	i16_last_step=> );

CASE fb_state_entry.i16_step OF
(*=======================================================*)
	INIT_OBJ:
		IF st_config.b_config_fertig THEN
			a_messbereich_1_oder_2 := FALSE;
			fb_state_entry.i16_next_step := INIT;
		END_IF

(*=======================================================*)
	INIT:
		IF fb_state_entry.E THEN
			fb_ton_wz.IN := FALSE;
			fb_ton_uez.IN := FALSE;
			fb_ton_quitt.IN := FALSE;
			st_ctrl_out.b_fehler := FALSE;
			st_ctrl_out.b_bereit := FALSE;
			st_ctrl_out.b_fertig := FALSE;
			a_start_messung := FALSE;
			i16_pin_nr := 0;
			sm_fehler_einpressmodus := FALSE;
			sm_aktkraft_groesser_maxkraft_aufnahme := FALSE;
			sm_aktkraft_groesser_maxkraft_einpressen := FALSE;
			sm_aktkraft_kleiner_minkraft_einpressen := FALSE;
			sm_kraft_weg_ausserhalb_huellkurve := FALSE;
			sm_fehler_analogwert_kraftmessdose := FALSE;
			sm_max_mb_ueberschritten := FALSE;
			sm_max_einstell_mb_ueberschritten := FALSE;
		END_IF

		(*-----------------------Weiterschaltbedingungen----------------------------*)
		IF st_ctrl_in.b_init THEN
			fb_state_entry.i16_next_step := BEREIT;
		END_IF

(*=======================================================*)
	BEREIT:
		IF fb_state_entry.E THEN
			st_ctrl_out.b_bereit := TRUE;
			st_ctrl_out.b_fertig := TRUE;
			i16_pin_nr := 0;
		END_IF

		(*-----------------------Weiterschaltbedingungen----------------------------*)
		IF st_ctrl_in.b_start THEN
			fb_state_entry.i16_next_step := 110;
		END_IF

(*=======================================================*)
	110:	(* Kraftmessung starten *)
		IF fb_state_entry.E THEN
			st_ctrl_out.b_fertig := FALSE;
			a_start_messung := TRUE;
			st_ausgabe.st_ergebnisse.lr_maxkraft_einpressen := 0;
			st_ausgabe.st_ergebnisse.lr_maxkraft_einpres_proHub:=0;
			st_ausgabe.st_ergebnisse.lr_ueberlaufkraft := 0;

			(* Löschen der Kraftwerte in den beiden IST-Einpresskurven *)
			FOR i16_ku_nr := 0  TO i_MAX_KURVEN BY 1DO
				FOR i16_mp_nr := 0  TO i_MAX_MESSPUNKTE BY 1DO
					st_ausgabe.st_kurve[i16_ku_nr].arr_kraft_ist[i16_mp_nr] := 0;
					st_ausgabe.st_kurve[i16_ku_nr].arr_weg_ist[i16_mp_nr] := 0;
				END_FOR
			END_FOR

			(* Löschen der Kraftwerte in allen Stützkurven*)
			IF st_einpressen.st_einstellungen.enu_modus = STUETZKURVE THEN
				FOR i16_ku_nr := 0  TO i_MAX_KURVEN BY 1DO
					FOR i16_mp_nr := 0  TO i_MAX_MESSPUNKTE BY 1DO
						st_ausgabe.st_kurve[i16_ku_nr].arr_kraft_stuetz[i16_mp_nr] := 0;
						st_ausgabe.st_kurve[i16_ku_nr].arr_weg_stuetz[i16_mp_nr] := 0;
					END_FOR
				END_FOR
			END_IF
		END_IF

		(* Hochzählen mit der Anzahl der bestückten Pins *)
		i16_pin_nr := ST_Virtuelle_Masterachse.i16_bestueckposzaehler;
		(* Abfrage Array-Grösse auf Überlauf *)
		IF i16_pin_nr > i_MAX_KURVEN THEN
			i16_pin_nr := 0;
		END_IF

		(* Die Messpunkte werden gradgenau aufgenommen und entsprechen deshalb den Winkelgraden der Bestückachse *)
		i16_mp_nr := ui_akt_pos_bestueckachse;

		CASE st_einpressen.st_einstellungen.enu_modus OF
			KEIN_MODUS:	(* Fehler Auswahl Einpressmodus *)
				sm_fehler_einpressmodus := TRUE;
				fb_state_entry.i16_next_step := FEHLER;

			FMAX:	(* Einpressen mit Überwachung auf Maximalkraft und Sicherheitsabfrage der Minimalkraft*)
				(*st_einpressen.st_einstellungen.lr_minkraft_einpressen := 12.0;*)
				IF  lr_kraft_n > st_ausgabe.st_ergebnisse.lr_maxkraft_einpressen THEN
					st_ausgabe.st_ergebnisse.lr_maxkraft_einpressen := lr_kraft_n;
				END_IF
				(* Fehlerfall: Voreingestellte Maximalkraft überschritten nur im Automatik Betrieb *)
				IF  gi16_betriebsart = AUTO AND lr_kraft_n > lr_help_maxkraft_einpressen THEN		(*st_einpressen.st_einstellungen.lr_maxkraft_einpressen*)
					sm_aktkraft_groesser_maxkraft_einpressen := TRUE;
					fb_state_entry.i16_next_step := FEHLER;
				END_IF

				(* Fehlerfall: Voreingestellte Minimalkraft unterschritten *)
				IF	lr_weg_grad =0 THEN
					st_ausgabe.st_ergebnisse.lr_maxkraft_einpres_proHub:=0;
				END_IF
				IF  lr_kraft_n > st_ausgabe.st_ergebnisse.lr_maxkraft_einpres_proHub THEN
					st_ausgabe.st_ergebnisse.lr_maxkraft_einpres_proHub:=lr_kraft_n;
				END_IF

				IF	gi16_betriebsart = AUTO AND
					st_einpressen.st_einstellungen.lr_minkraft_einpressen > 0 AND
					nockenschaltwerk_bestueckachse.fb.arr_spur[SP_BESTUECKSCHIEBERHUB ] AND
					st_ausgabe.st_ergebnisse.lr_maxkraft_einpres_proHub < st_einpressen.st_einstellungen.lr_minkraft_einpressen	THEN
					i16_merker:=i16_merker+1;
					(*	sm_aktkraft_kleiner_minkraft_einpressen := TRUE;
						fb_state_entry.i16_next_step := FEHLER;*)
				END_IF

				(* Aufzeichnen der Überlaufkraft nach einem Einpressfehler *)
				IF  lr_kraft_n > st_ausgabe.st_ergebnisse.lr_ueberlaufkraft THEN
					st_ausgabe.st_ergebnisse.lr_ueberlaufkraft := lr_kraft_n;
				END_IF

			FMIN_FMAX:	(* Einpressen mit Überwachung von Minimal- und Maximalkraft. Der Weg spielt hier keine Rolle! *)
				(* Aktuelle Kraft gradgenau einlesen *)
				IF st_ausgabe.st_kurve[i16_pin_nr].arr_kraft_ist[i16_mp_nr] = 0 THEN
					(* Einmalig den aktuellen Kraftwert eintragen, wenn Messpunkt im Array noch leer ist *)
					st_ausgabe.st_kurve[i16_pin_nr].arr_kraft_ist[i16_mp_nr] := lr_kraft_n;
				END_IF

				(* Aufnehmen der maximal aufgetretenen Kraft *)
				IF st_ausgabe.st_kurve[i16_pin_nr].arr_kraft_ist[i16_mp_nr] > st_ausgabe.st_ergebnisse.lr_maxkraft_einpressen THEN
					st_ausgabe.st_ergebnisse.lr_maxkraft_einpressen := st_ausgabe.st_kurve[i16_pin_nr].arr_kraft_ist[i16_mp_nr];
				END_IF

				(* Fehlerfall: Überwachen der Maximalkraft beim Aufnahmehub *)
				IF 	nockenschaltwerk_bestueckachse.fb.arr_spur[SP_AUFNAHMEHUB ] AND
					st_ausgabe.st_kurve[i16_pin_nr].arr_kraft_ist[i16_mp_nr] > 0
					THEN
						IF st_ausgabe.st_kurve[i16_pin_nr].arr_kraft_ist[i16_mp_nr] > st_einpressen.st_einstellungen.lr_maxkraft_aufnahme THEN
							st_einpressen.st_einstellungen.lr_maxkraft_aufnahme := st_ausgabe.st_kurve[i16_pin_nr].arr_kraft_ist[i16_mp_nr];
							sm_aktkraft_groesser_maxkraft_aufnahme := TRUE;
							fb_state_entry.i16_next_step := FEHLER;
						END_IF
				END_IF

				(* Fehlerfall: Überwachen der Maximalkraft beim Auftreffen des Pins auf den Isolierkörper *)
				IF 	nockenschaltwerk_bestueckachse.fb.arr_spur[SP_EINPRESSHUB ] AND
					st_ausgabe.st_kurve[i16_pin_nr].arr_kraft_ist[i16_mp_nr] > 0
					THEN
						IF st_ausgabe.st_kurve[i16_pin_nr].arr_kraft_ist[i16_mp_nr] > st_einpressen.st_einstellungen.lr_maxkraft_einpressen THEN
							st_einpressen.st_einstellungen.lr_maxkraft_einpressen := st_ausgabe.st_kurve[i16_pin_nr].arr_kraft_ist[i16_mp_nr];
							sm_aktkraft_groesser_maxkraft_einpressen := TRUE;
							fb_state_entry.i16_next_step := FEHLER;
						END_IF
				END_IF

				(* Fehlerfall: Überwachen der Minimalkraft beim Einpresshub *)
				IF 	nockenschaltwerk_bestueckachse.fb.arr_spur[SP_MIN_KRAFT_EINPRESSEN ] AND
					st_ausgabe.st_kurve[i16_pin_nr].arr_kraft_ist[i16_mp_nr] > 0
					THEN
						IF st_ausgabe.st_kurve[i16_pin_nr].arr_kraft_ist[i16_mp_nr] < st_einpressen.st_einstellungen.lr_minkraft_einpressen THEN
							st_einpressen.st_einstellungen.lr_minkraft_einpressen := st_ausgabe.st_kurve[i16_pin_nr].arr_kraft_ist[i16_mp_nr];
							sm_aktkraft_kleiner_minkraft_einpressen := TRUE;
							fb_state_entry.i16_next_step := FEHLER;
						END_IF
				END_IF

			HUELLKURVE:	(* Einpressen mit Hüllkurve um Stützkurve*)
				(* Aktuelle Kraft in die Ist-Kurve einlesen *)
				IF st_ausgabe.st_kurve[i16_pin_nr].arr_kraft_ist[i16_mp_nr] = 0 THEN
					(* Einmalig den aktuellen Kraftwert eintragen, wenn Messpunkt im Array noch leer ist *)
					st_ausgabe.st_kurve[i16_pin_nr].arr_kraft_ist[i16_mp_nr] := lr_kraft_n;
				END_IF
				(* Aktuellen Weg in die Ist-Kurve einlesen, wobei in diesem Fall das Arrayelement dem aktuellen Winkel entspricht. *)
				IF st_ausgabe.st_kurve[i16_pin_nr].arr_weg_ist[i16_mp_nr] = 0 THEN
					(* Einmalig den aktuellen Wegwert eintragen, wenn Messpunkt im Array noch leer ist *)
					st_ausgabe.st_kurve[i16_pin_nr].arr_weg_ist[i16_mp_nr] := lr_weg_grad;
				END_IF

				(* Toleranzabfrage und Fehlerauswertung *)
				IF st_ausgabe.st_kurve[i16_pin_nr].arr_kraft_ist[i16_mp_nr] > 0 AND st_ausgabe.st_kurve[i16_pin_nr].arr_weg_ist[i16_mp_nr] > 0 THEN
					b_kraft_weg_in_mp_ok := FALSE;
					(* Werte sind gültig -> Abfrage , ob Kraft und Weg im Toleranzrechteck liegen. *)
					FOR i16_mp_nr := 0  TO i_MAX_MESSPUNKTE BY 1DO
						IF	st_ausgabe.st_kurve[i16_pin_nr].arr_kraft_ist[i16_mp_nr] >= (st_ausgabe.st_kurve[i16_pin_nr].arr_kraft_ist[i16_mp_nr] - st_einpressen.st_einstellungen.lr_delta_kraft) AND
							st_ausgabe.st_kurve[i16_pin_nr].arr_kraft_ist[i16_mp_nr] <= (st_ausgabe.st_kurve[i16_pin_nr].arr_kraft_ist[i16_mp_nr] + st_einpressen.st_einstellungen.lr_delta_kraft) AND
							st_ausgabe.st_kurve[i16_pin_nr].arr_weg_ist[i16_mp_nr] >= (st_ausgabe.st_kurve[i16_pin_nr].arr_weg_ist[i16_mp_nr] - st_einpressen.st_einstellungen.lr_delta_weg) AND
							st_ausgabe.st_kurve[i16_pin_nr].arr_weg_ist[i16_mp_nr] <= (st_ausgabe.st_kurve[i16_pin_nr].arr_weg_ist[i16_mp_nr] + st_einpressen.st_einstellungen.lr_delta_weg)
							THEN
								b_kraft_weg_in_mp_ok := TRUE;
								EXIT;
						ELSE
							b_kraft_weg_in_mp_ok := FALSE;
						END_IF
					END_FOR

					(* Fehlerfall: Aktueller Messpunkt liegt mit seiner Kraft oder seinem Weg nicht im Toleranzrechteck *)
					IF NOT b_kraft_weg_in_mp_ok THEN
						sm_kraft_weg_ausserhalb_huellkurve := TRUE;
						fb_state_entry.i16_next_step := FEHLER;
					END_IF
				END_IF

			STUETZKURVE:	(* Einlernen der Stützkurve *)
				(* Aktuelle Kraft in die Stuetzkurve einlesen *)
				IF st_ausgabe.st_kurve[i16_pin_nr].arr_kraft_stuetz[i16_mp_nr] = 0 THEN
					(* Einmalig den aktuellen Kraftwert eintragen, wenn Messpunkt im Array noch leer ist *)
					st_ausgabe.st_kurve[i16_pin_nr].arr_kraft_stuetz[i16_mp_nr] := lr_kraft_n;
				END_IF
				(* Aktuellen Weg in die Stuetzkurve einlesen, wobei in diesem Fall das Arrayelement dem aktuellen Winkel entspricht. *)
				IF st_ausgabe.st_kurve[i16_pin_nr].arr_weg_stuetz[i16_mp_nr] = 0 THEN
					(* Einmalig den aktuellen Wegwert eintragen, wenn Messpunkt im Array noch leer ist *)
					st_ausgabe.st_kurve[i16_pin_nr].arr_weg_stuetz[i16_mp_nr] := lr_weg_grad;
				END_IF
		END_CASE

		(* Manuelle Messbereichsumschaltung anhand des Einstellwertes für Maximalkraft beim Einpressen. *)
		IF gst_datensatz.st_band.st_einpressen.st_einstellungen.lr_maxkraft_einpressen > (i_KRAFTFAKTOR_MB1 * 0.75) THEN
			a_messbereich_1_oder_2 := TRUE;
		ELSE
			(* Automatische Messbereichsumschaltung, wenn die maximale Einpresskraft 75% des Messbereichsendwertes überschreitet. *)
			IF st_ausgabe.st_ergebnisse.lr_maxkraft_einpressen > (i_KRAFTFAKTOR_MB1 * 0.75) THEN
				a_messbereich_1_oder_2 := TRUE;
			END_IF
		END_IF

		(*-----------------------Weiterschaltbedingungen----------------------------*)
		IF NOT st_ctrl_in.b_start THEN
			(* Messbereichsanpassung nur, wenn die Krafteinstellung für maximale Einpresskraft es erlaubt. *)
			IF gst_datensatz.st_band.st_einpressen.st_einstellungen.lr_maxkraft_einpressen < (i_KRAFTFAKTOR_MB1 * 0.75) THEN
				(* Automatische Messbereichsumschaltung, wenn die maximale Einpresskraft 50% des Messbereichsendwertes unterschreitet. *)
				IF st_ausgabe.st_ergebnisse.lr_maxkraft_einpressen < (i_KRAFTFAKTOR_MB1 * 0.5) THEN
					a_messbereich_1_oder_2 := FALSE;
				END_IF
			END_IF
			a_start_messung := FALSE;
			fb_state_entry.i16_next_step := BEREIT;
		END_IF

(*=======================================================*)
	FEHLER:
		IF fb_state_entry.E THEN
			st_ctrl_out.b_fehler := TRUE;
			fb_ton_quitt.IN := FALSE;
		END_IF

		(* Aufzeichnen der Überlaufkraft nach einem Einpressfehler *)
		IF  lr_kraft_n > st_ausgabe.st_ergebnisse.lr_ueberlaufkraft THEN
			st_ausgabe.st_ergebnisse.lr_ueberlaufkraft := lr_kraft_n;
		END_IF

		(*-----------------------Weiterschaltbedingungen----------------------------*)
		IF st_ctrl_in.b_quitt AND NOT fb_state_entry.E THEN
			st_ctrl_out.b_fehler := FALSE;
			fb_ton_quitt.IN := TRUE;
		END_IF

		IF fb_ton_quitt.Q THEN
			fb_ton_quitt.IN := FALSE;
			fb_state_entry.i16_next_step := INIT;
		END_IF

(*=======================================================*)
	STOP:
		IF fb_state_entry.E THEN
			fb_ton_quitt.IN := FALSE;
		END_IF

		(*-----------------------Weiterschaltbedingungen----------------------------*)
		IF st_ctrl_in.b_quitt AND NOT fb_state_entry.E THEN
			fb_ton_quitt.IN := TRUE;
		END_IF

		IF fb_ton_quitt.Q THEN
			fb_ton_quitt.IN := FALSE;
			fb_state_entry.i16_next_step := INIT;
		END_IF
END_CASE

fb_state_entry(
	i16_next_step:= ,
	i16_pos:= 2,
	s_debugtext:= ,
	E=> , 
	X=> ,
	i16_step=> ,
	i16_last_step=> );

(* Fehlermeldungen und Betriebsmeldungen ab dem Startindex in die globalen Meldungsarrays schreiben *)
garr_stoermeldungen[st_config.i16_meld_startindex + 0] := sm_fehler_einpressmodus;
garr_stoermeldungen[st_config.i16_meld_startindex + 1] := sm_aktkraft_groesser_maxkraft_aufnahme;
garr_stoermeldungen[st_config.i16_meld_startindex + 2] := sm_aktkraft_groesser_maxkraft_einpressen;
garr_stoermeldungen[st_config.i16_meld_startindex + 3] := sm_aktkraft_kleiner_minkraft_einpressen;
garr_stoermeldungen[st_config.i16_meld_startindex + 4] := sm_kraft_weg_ausserhalb_huellkurve;
garr_stoermeldungen[st_config.i16_meld_startindex + 5] := sm_fehler_analogwert_kraftmessdose;
garr_stoermeldungen[st_config.i16_meld_startindex + 6] := sm_max_mb_ueberschritten;
garr_stoermeldungen[st_config.i16_meld_startindex + 7] := sm_max_einstell_mb_ueberschritten;
garr_stoermeldungen[st_config.i16_meld_startindex + 8] := FALSE;
garr_stoermeldungen[st_config.i16_meld_startindex + 9] := FALSE;
garr_stoermeldungen[st_config.i16_meld_startindex + 10] := FALSE;
garr_stoermeldungen[st_config.i16_meld_startindex + 11] := FALSE;
garr_stoermeldungen[st_config.i16_meld_startindex + 12] := FALSE;
garr_stoermeldungen[st_config.i16_meld_startindex + 13] := FALSE;
garr_stoermeldungen[st_config.i16_meld_startindex + 14] := FALSE;
garr_stoermeldungen[st_config.i16_meld_startindex + 15] := FALSE;
garr_stoermeldungen[st_config.i16_meld_startindex + 16] := FALSE;
garr_stoermeldungen[st_config.i16_meld_startindex + 17] := FALSE;
garr_stoermeldungen[st_config.i16_meld_startindex + 18] := FALSE;
garr_stoermeldungen[st_config.i16_meld_startindex + 19] := FALSE;

garr_betriebsmeldungen[st_config.i16_meld_startindex + 0] := FALSE;
garr_betriebsmeldungen[st_config.i16_meld_startindex + 1] := FALSE;
garr_betriebsmeldungen[st_config.i16_meld_startindex + 2] := FALSE;
garr_betriebsmeldungen[st_config.i16_meld_startindex + 3] := FALSE;
garr_betriebsmeldungen[st_config.i16_meld_startindex + 4] := FALSE;
garr_betriebsmeldungen[st_config.i16_meld_startindex + 5] := FALSE;
garr_betriebsmeldungen[st_config.i16_meld_startindex + 6] := FALSE;
garr_betriebsmeldungen[st_config.i16_meld_startindex + 7] := FALSE;
garr_betriebsmeldungen[st_config.i16_meld_startindex + 8] := FALSE;
garr_betriebsmeldungen[st_config.i16_meld_startindex + 9] := FALSE;
garr_betriebsmeldungen[st_config.i16_meld_startindex + 10] := FALSE;
garr_betriebsmeldungen[st_config.i16_meld_startindex + 11] := FALSE;
garr_betriebsmeldungen[st_config.i16_meld_startindex + 12] := FALSE;
garr_betriebsmeldungen[st_config.i16_meld_startindex + 13] := FALSE;
garr_betriebsmeldungen[st_config.i16_meld_startindex + 14] := FALSE;
garr_betriebsmeldungen[st_config.i16_meld_startindex + 15] := FALSE;
garr_betriebsmeldungen[st_config.i16_meld_startindex + 16] := FALSE;
garr_betriebsmeldungen[st_config.i16_meld_startindex + 17] := FALSE;
garr_betriebsmeldungen[st_config.i16_meld_startindex + 18] := FALSE;
garr_betriebsmeldungen[st_config.i16_meld_startindex + 19] := FALSE;
END_PROGRAM

(* POU Gemeinsamkeiten17xx/Oeler/ST_Einzelbandoeler, ST *)
PROGRAM ST_Einzelbandoeler
VAR_INPUT
	st_config						: struct_config;
	st_ctrl_in						: struct_ctrl_in;
	b_ot_spur					: BOOL;
END_VAR
VAR_IN_OUT
	st_visu						: struct_oeler_visu;
	st_oelerdaten					: struct_oeler_retain;
END_VAR
VAR_OUTPUT
	st_ctrl_out					: struct_ctrl_out;
END_VAR
VAR
	fb_ton_quitt					: TON;
	dt_datum_uhrzeit_letzte_oelung	: DT;
	fb_state_entry					: ST_StateEntry;
	t_delta_zeitraum				: TIME := t#5h;
	a_ventil			 			AT %Q* : BOOL;
	e_fuellstand					AT %I* : BOOL;
	sm_fuellstand_oeler			: BOOL := FALSE;
	fb_ton_oelzeit					: TON;
	fb_r_trig_start_oelen			: R_TRIG;
	fb_r_trig_hubimpuls			: R_TRIG;

	fb_r_trig_ibn_handoelen		: R_TRIG;
	fb_ton_ibn_handoelen			: TON;
	b_ibn_handoelen				: BOOL := FALSE;
END_VAR
(* Bandöler mit Füllstandsabfrage und Zwangs- und Stillstandsölung *)
(* Oeler Impuls generieren *)
fb_ton_oelzeit(IN:= , PT:= , Q=> , ET=> );
fb_ton_quitt(IN:= , PT:= t#100ms, Q=> , ET=> );

(* Hubimpuls *)
fb_r_trig_hubimpuls(CLK:= b_ot_spur, Q=> );

(* Inbetriebnahme *)
fb_r_trig_ibn_handoelen(CLK:= b_ibn_handoelen, Q=> );
fb_ton_ibn_handoelen(IN:= , PT:= t#1s, Q=> , ET=> );
IF fb_r_trig_ibn_handoelen.Q THEN
	fb_ton_ibn_handoelen.IN := TRUE;
ELSE
	IF fb_ton_ibn_handoelen.Q THEN
		b_ibn_handoelen := FALSE;
	 	fb_ton_ibn_handoelen.IN := FALSE;
	END_IF
END_IF

(* =======================================Toplevel========================================== *)
IF fb_state_entry.i16_next_step > INIT AND fb_state_entry.i16_next_step < FEHLER THEN
	IF fb_state_entry.i16_next_step < STOP THEN
		IF st_ctrl_in.b_stop THEN
			fb_state_entry.i16_next_step := STOP;
		END_IF
	END_IF
END_IF

(* Prüfe auf neue Intervalvorgabe *)
IF st_config.b_station_aktiv AND st_oelerdaten.i32_neue_intervallvorgabe <> st_oelerdaten.i32_alte_intervallvorgabe THEN
	st_oelerdaten.i32_alte_intervallvorgabe := st_oelerdaten.i32_neue_intervallvorgabe;
	st_oelerdaten.i32_aktueller_stand := st_oelerdaten.i32_neue_intervallvorgabe;
END_IF

(* ==================================Schrittkette================================ *)
fb_state_entry(
	i16_next_step:= , 
	i16_pos:= 1,
	s_debugtext:= ,
	E=> ,
	X=> , 
	i16_step=> ,
	i16_last_step=> );

CASE fb_state_entry.i16_step OF
(*=======================================================*)
	INIT_OBJ:
		IF st_config.b_config_fertig THEN
			fb_state_entry.i16_next_step := INIT;
		END_IF
		
(*=======================================================*)
	INIT:
		IF fb_state_entry.E THEN
			st_ctrl_out.b_fehler := FALSE;
			st_ctrl_out.b_bereit := FALSE;
			st_ctrl_out.b_fertig := FALSE;
			fb_ton_oelzeit.IN := FALSE;
			fb_ton_ibn_handoelen.IN := FALSE;
			fb_ton_quitt.IN := FALSE;
			a_ventil := FALSE;
			sm_fuellstand_oeler := FALSE;
		END_IF

		(*-----------------------Weiterschaltbedingungen----------------------------*)
		IF st_ctrl_in.b_init THEN
			IF st_config.b_station_aktiv THEN
				fb_state_entry.i16_next_step := 20;
			ELSE
				fb_state_entry.i16_next_step := BEREIT;
			END_IF
		END_IF

(*=======================================================*)
	20: (* Abfrage Datum / Uhrzeit wegen Ölen nach Stillstand*)

		(*-----------------------Weiterschaltbedingungen----------------------------*)
		IF (gdt_system_time - dt_datum_uhrzeit_letzte_oelung) > t_delta_zeitraum THEN
			fb_ton_oelzeit.PT := st_oelerdaten.t_oelzeit_nach_stillstand;
			fb_state_entry.i16_next_step := 30;
		ELSE
			fb_state_entry.i16_next_step := BEREIT;
		END_IF

(*=======================================================*)
	30: (* Ölen nach Stillstand *)
		IF fb_state_entry.E THEN
			dt_datum_uhrzeit_letzte_oelung := gdt_system_time;	(* Merken, dass geölt wurde *)
			fb_ton_oelzeit.IN := TRUE;
			a_ventil := TRUE;
		END_IF

		(*-----------------------Weiterschaltbedingungen----------------------------*)
		IF  fb_ton_oelzeit.Q THEN
			fb_ton_oelzeit.IN := FALSE;
			a_ventil := FALSE;
			fb_state_entry.i16_next_step := BEREIT;
		END_IF

(*=======================================================*)
	BEREIT:
		IF fb_state_entry.E THEN
			st_ctrl_out.b_bereit := TRUE;
		END_IF

		IF st_config.b_station_aktiv THEN
			(* Zähle Hübe *)
			IF fb_r_trig_hubimpuls.Q THEN
				(* Von der Intervallvorgabe wird runter gezählt bis Null. Dann kommt der Ölimpuls *)
				st_oelerdaten.i32_aktueller_stand := st_oelerdaten.i32_aktueller_stand - 1;
			END_IF
			(* Überwachung Füllstand *)
			IF NOT e_fuellstand THEN
				sm_fuellstand_oeler := TRUE;
				fb_state_entry.i16_next_step := FEHLER;
			END_IF

			(*-----------------------Weiterschaltbedingungen----------------------------*)
			IF  st_oelerdaten.i32_aktueller_stand <= 0 OR st_visu.b_handoelen OR fb_r_trig_ibn_handoelen.Q THEN
				st_visu.b_handoelen := FALSE;
				fb_ton_oelzeit.PT := st_oelerdaten.t_ventiloeffnungszeit;
				fb_state_entry.i16_next_step := 110;
			END_IF
		END_IF

(*=======================================================*)
	110: (* Ölen *)
		IF fb_state_entry.E THEN
			dt_datum_uhrzeit_letzte_oelung := gdt_system_time;	(* Merken wann das letze mal geölt wurde *)
			IF st_oelerdaten.i32_neue_intervallvorgabe <= 0 THEN
				 st_oelerdaten.i32_neue_intervallvorgabe := 100;	(* Verhindere Dauerölung, wenn in den WKZ-Ölerdaten noch 0 drin steht *)
			END_IF
			st_oelerdaten.i32_aktueller_stand := st_oelerdaten.i32_neue_intervallvorgabe;
			fb_ton_oelzeit.IN := TRUE;
			a_ventil := TRUE;
		END_IF

		(* Zähle Hübe *)
		IF fb_r_trig_hubimpuls.Q THEN
			(* Von der Intervallvorgabe wird runter gezählt bis Null. Dann kommt der Ölimpuls *)
			st_oelerdaten.i32_aktueller_stand := st_oelerdaten.i32_aktueller_stand - 1;
		END_IF

		(*-----------------------Weiterschaltbedingungen----------------------------*)
		IF  fb_ton_oelzeit.Q THEN
			fb_ton_oelzeit.IN := FALSE;
			a_ventil := FALSE;
			fb_state_entry.i16_next_step := BEREIT;
		END_IF

(*=======================================================*)
	FEHLER:
		IF fb_state_entry.E THEN
			st_ctrl_out.b_fehler := TRUE;
			a_ventil := FALSE;
			fb_ton_quitt.IN := FALSE;
		END_IF

		(*-----------------------Weiterschaltbedingungen----------------------------*)
		IF st_ctrl_in.b_quitt AND NOT fb_state_entry.E THEN
			st_ctrl_out.b_fehler := FALSE;
			fb_ton_quitt.IN := TRUE;
		END_IF

		IF fb_ton_quitt.Q THEN
			fb_ton_quitt.IN := FALSE;
			fb_state_entry.i16_next_step := INIT;
		END_IF

(*=======================================================*)
	STOP:
		IF fb_state_entry.E THEN
			a_ventil := FALSE;
			fb_ton_quitt.IN := FALSE;
		END_IF

		(*-----------------------Weiterschaltbedingungen----------------------------*)
		IF st_ctrl_in.b_quitt AND NOT fb_state_entry.E THEN
			fb_ton_quitt.IN := TRUE;
		END_IF

		IF fb_ton_quitt.Q THEN
			fb_ton_quitt.IN := FALSE;
			fb_state_entry.i16_next_step := INIT;
		END_IF
END_CASE

fb_state_entry(
	i16_next_step:= , 
	i16_pos:= 2,
	s_debugtext:= ,
	E=> ,
	X=> , 
	i16_step=> ,
	i16_last_step=> );

IF st_config.b_config_fertig THEN
	(* Fehlermeldungen und Betriebsmeldungen ab dem Startindex in die globalen Meldungsarrays schreiben *)
	garr_stoermeldungen[st_config.i16_meld_startindex + 0] := sm_fuellstand_oeler;
	garr_stoermeldungen[st_config.i16_meld_startindex + 1] := FALSE;
	garr_stoermeldungen[st_config.i16_meld_startindex + 2] := FALSE;
	garr_stoermeldungen[st_config.i16_meld_startindex + 3] := FALSE;
	garr_stoermeldungen[st_config.i16_meld_startindex + 4] := FALSE;
	garr_stoermeldungen[st_config.i16_meld_startindex + 5] := FALSE;
	garr_stoermeldungen[st_config.i16_meld_startindex + 6] := FALSE;
	garr_stoermeldungen[st_config.i16_meld_startindex + 7] := FALSE;
	garr_stoermeldungen[st_config.i16_meld_startindex + 8] := FALSE;
	garr_stoermeldungen[st_config.i16_meld_startindex + 9] := FALSE;
	garr_stoermeldungen[st_config.i16_meld_startindex + 10] := FALSE;
	garr_stoermeldungen[st_config.i16_meld_startindex + 11] := FALSE;
	garr_stoermeldungen[st_config.i16_meld_startindex + 12] := FALSE;
	garr_stoermeldungen[st_config.i16_meld_startindex + 13] := FALSE;
	garr_stoermeldungen[st_config.i16_meld_startindex + 14] := FALSE;
	garr_stoermeldungen[st_config.i16_meld_startindex + 15] := FALSE;
	garr_stoermeldungen[st_config.i16_meld_startindex + 16] := FALSE;
	garr_stoermeldungen[st_config.i16_meld_startindex + 17] := FALSE;
	garr_stoermeldungen[st_config.i16_meld_startindex + 18] := FALSE;
	garr_stoermeldungen[st_config.i16_meld_startindex + 19] := FALSE;
	
	garr_betriebsmeldungen[st_config.i16_meld_startindex + 0] := FALSE;
	garr_betriebsmeldungen[st_config.i16_meld_startindex + 1] := FALSE;
	garr_betriebsmeldungen[st_config.i16_meld_startindex + 2] := FALSE;
	garr_betriebsmeldungen[st_config.i16_meld_startindex + 3] := FALSE;
	garr_betriebsmeldungen[st_config.i16_meld_startindex + 4] := FALSE;
	garr_betriebsmeldungen[st_config.i16_meld_startindex + 5] := FALSE;
	garr_betriebsmeldungen[st_config.i16_meld_startindex + 6] := FALSE;
	garr_betriebsmeldungen[st_config.i16_meld_startindex + 7] := FALSE;
	garr_betriebsmeldungen[st_config.i16_meld_startindex + 8] := FALSE;
	garr_betriebsmeldungen[st_config.i16_meld_startindex + 9] := FALSE;
	garr_betriebsmeldungen[st_config.i16_meld_startindex + 10] := FALSE;
	garr_betriebsmeldungen[st_config.i16_meld_startindex + 11] := FALSE;
	garr_betriebsmeldungen[st_config.i16_meld_startindex + 12] := FALSE;
	garr_betriebsmeldungen[st_config.i16_meld_startindex + 13] := FALSE;
	garr_betriebsmeldungen[st_config.i16_meld_startindex + 14] := FALSE;
	garr_betriebsmeldungen[st_config.i16_meld_startindex + 15] := FALSE;
	garr_betriebsmeldungen[st_config.i16_meld_startindex + 16] := FALSE;
	garr_betriebsmeldungen[st_config.i16_meld_startindex + 17] := FALSE;
	garr_betriebsmeldungen[st_config.i16_meld_startindex + 18] := FALSE;
	garr_betriebsmeldungen[st_config.i16_meld_startindex + 19] := FALSE;
END_IF
END_PROGRAM

(* POU Gemeinsamkeiten17xx/Haspel/Mehrfach/ST_Haspel_Kontroller_4H, ST *)
PROGRAM ST_Haspel_Kontroller_4H
VAR_INPUT
	t_abschaltzeit_motor			: TIME;
	b_drehrichtung_antrieb_links	: BOOL;
	st_config						: struct_config;
	e_druckwaechter				: BOOL;
	e_steuerung_ein				: BOOL;
	st_ctrl_in						: struct_ctrl_in;
	haspel1_ctrl_in				: struct_ctrl_out;
	haspel2_ctrl_in				: struct_ctrl_out;
	haspel3_ctrl_in				: struct_ctrl_out;
	haspel4_ctrl_in				: struct_ctrl_out;
END_VAR
VAR_IN_OUT
	st_visu						: struct_visu;
END_VAR
VAR_OUTPUT
	st_ctrl_out					: struct_ctrl_out;
	haspel1_ctrl_out				: struct_ctrl_in;
	haspel2_ctrl_out				: struct_ctrl_in;
	haspel3_ctrl_out				: struct_ctrl_in;
	haspel4_ctrl_out				: struct_ctrl_in;
END_VAR
VAR
	fb_ton_wz					: TON;
	fb_ton_uez					: TON;
	fb_ton_vz					: TON;
	fb_ton_quitt					: TON;
	fb_tof_motor					: TOF;
	b_motor_laeuft				: BOOL := FALSE;
	fb_state_entry					: ST_StateEntry;
	a_motor_drehrichtung_rechts	AT %Q* : BOOL;
	a_motor_drehrichtung_links		AT %Q* : BOOL;
END_VAR
(* Zeiten *)
fb_ton_wz(IN:= , PT:= , Q=>  , ET=> );
fb_ton_uez(IN:= , PT:= , Q=>  , ET=> );
fb_ton_vz(IN:= , PT:= , Q=>  , ET=> );
fb_tof_motor(IN:= , PT:= t_abschaltzeit_motor, Q=> , ET=> );
fb_ton_quitt(IN:= , PT:= t#100ms, Q=> , ET=> );

b_motor_laeuft := a_motor_drehrichtung_links OR a_motor_drehrichtung_rechts;

(* Bandende von Haspel rechts bzw. links *)
IF	(gi16_betriebsart = AUTO OR gi16_betriebsart = TIPPEN) AND
 	(haspel1_ctrl_in.b_bandende OR
	haspel2_ctrl_in.b_bandende OR
	haspel3_ctrl_in.b_bandende OR
	haspel4_ctrl_in.b_bandende)
	THEN
		st_ctrl_out.b_bandende := TRUE;
ELSE
		st_ctrl_out.b_bandende := FALSE;
END_IF

(* Toplevel *)
IF fb_state_entry.i16_next_step > INIT AND fb_state_entry.i16_next_step < FEHLER THEN
	IF fb_state_entry.i16_next_step < STOP THEN
		IF st_ctrl_in.b_stop THEN
			fb_state_entry.i16_next_step := STOP;
		END_IF
	END_IF
	IF 	haspel1_ctrl_in.b_fehler OR
		haspel2_ctrl_in.b_fehler OR
		haspel3_ctrl_in.b_fehler OR
		haspel4_ctrl_in.b_fehler
		THEN
			fb_state_entry.i16_next_step := FEHLER;
	END_IF
END_IF

(* ==================================Schrittkette================================ *)
fb_state_entry(
	i16_next_step:= , 
	i16_pos:= 1,
	s_debugtext:= ,
	E=> ,
	X=> , 
	i16_step=> ,
	i16_last_step=> );

CASE fb_state_entry.i16_step OF
(*=======================================================*)
	INIT_OBJ:
		IF st_config.b_config_fertig THEN
			fb_state_entry.i16_next_step := INIT;
		END_IF

(*=======================================================*)
	INIT:
		IF fb_state_entry.E THEN
			fb_ton_wz.IN := FALSE;
			fb_ton_uez.IN	:= FALSE;
			fb_ton_vz.IN := FALSE;
			fb_ton_quitt.IN := FALSE;
			a_motor_drehrichtung_links 	:= FALSE;
			a_motor_drehrichtung_rechts := FALSE;
			st_ctrl_out.b_fehler := FALSE;
			st_ctrl_out.b_bereit := FALSE;
			st_ctrl_out.b_fertig := FALSE;
			haspel1_ctrl_out.b_init := FALSE;
			haspel2_ctrl_out.b_init := FALSE;
			haspel3_ctrl_out.b_init := FALSE;
			haspel4_ctrl_out.b_init := FALSE;
		END_IF

		(*-----------------------Weiterschaltbedingungen----------------------------*)
		IF st_ctrl_in.b_init THEN
			haspel1_ctrl_out.b_quitt := FALSE;
			haspel2_ctrl_out.b_quitt := FALSE;
			haspel3_ctrl_out.b_quitt := FALSE;
			haspel4_ctrl_out.b_quitt := FALSE;
			fb_state_entry.i16_next_step :=20;
		END_IF

